// /Chiller_2_Values
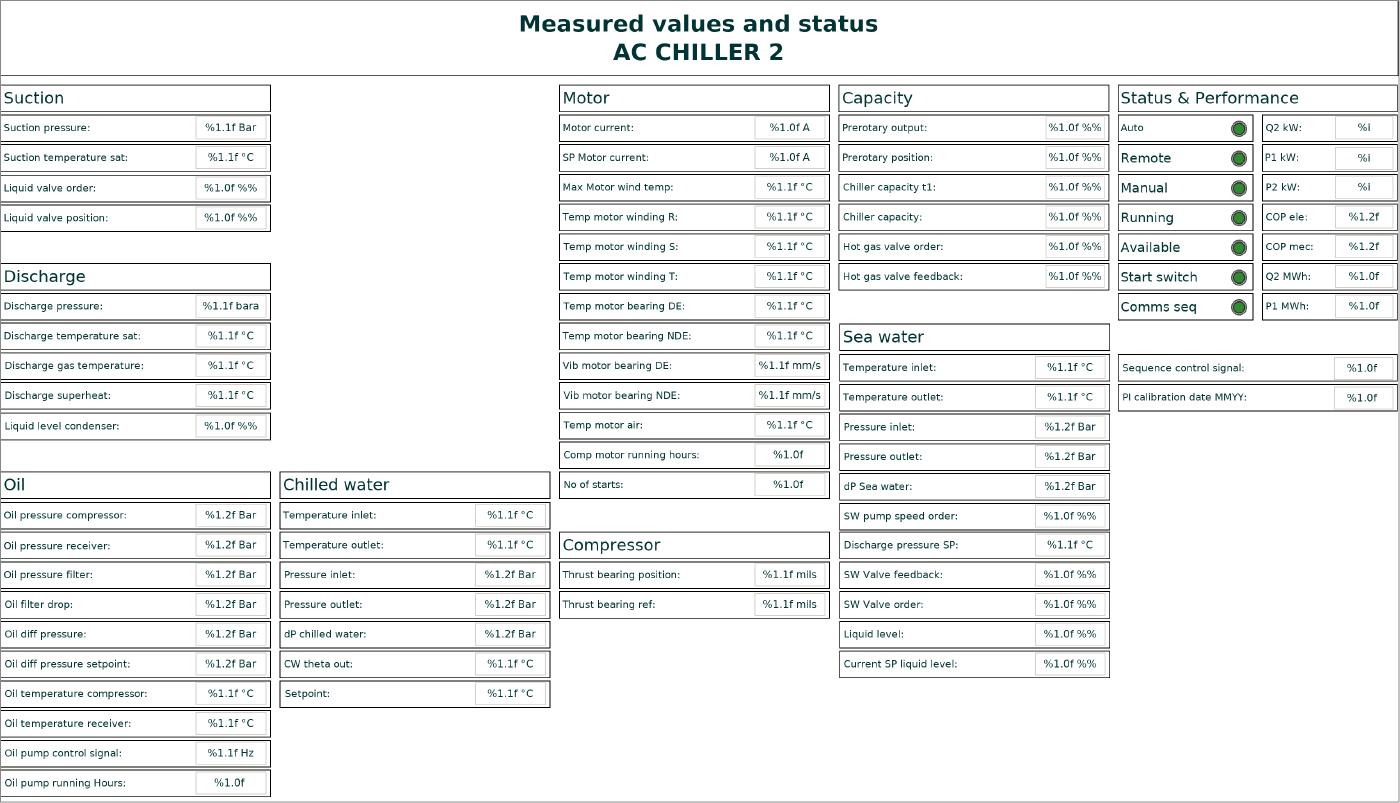
VISUALIZATION Chiller_2_Values  // 1553x891
    Rectangle (0,0 1551x84)
    Label (319,7 912x70), "Measured values and status AC CHILLER 2"
    Rectangle (0,94 300x30)
    Label (1,94 215x30), "Suction"
    Rectangle (0,127 300x30)
    Label (1,122 208x40), "Suction pressure:"
    Textfield (217,129 78x25), "%1.1f Bar", tooltip "Chiller_2.Press_suction_compr", text variable: Chiller_2.Press_suction_compr
        p4168582468: Chiller_2.Press_suction_compr
    Rectangle (0,160 300x30)
    Label (1,155 209x40), "Suction temperature sat:"
    Textfield (217,162 78x25), "%1.1f °C", tooltip "Chiller_2.Suction_saturated_temp", text variable: Chiller_2.Suction_saturated_temp
        p4168582468: Chiller_2.Suction_saturated_temp
    Rectangle (0,194 300x30)
    Label (1,189 211x40), "Liquid valve order:"
    Textfield (217,196 78x25), "%1.0f %%", tooltip "Chiller_2.Liquid_valve_output", text variable: Chiller_2.Liquid_valve_output
        p4168582468: Chiller_2.Liquid_valve_output
    Rectangle (0,227 300x30)
    Label (1,222 216x40), "Liquid valve position:"
    Textfield (217,229 78x25), "%1.0f %%", tooltip "Chiller_2.Feedback_liquid_valve", text variable: Chiller_2.Feedback_liquid_valve
        p4168582468: Chiller_2.Feedback_liquid_valve
    Rectangle (930,94 300x30)
    Label (931,94 162x30), "Capacity"
    Rectangle (930,127 300x30)
    Label (931,126 174x32), "Prerotary output:"
    Textfield (1160,129 65x25), "%1.0f %%", tooltip "Chiller_2.Prerotary_output", text variable: Chiller_2.Prerotary_output
        p4168582468: Chiller_2.Prerotary_output
    Rectangle (930,160 300x30)
    Label (931,159 173x32), "Prerotary position:"
    Textfield (1160,162 65x25), "%1.0f %%", tooltip "Chiller_2.Feedback_PRV", text variable: Chiller_2.Feedback_PRV
        p4168582468: Chiller_2.Feedback_PRV
    Rectangle (930,259 300x30)
    Label (932,258 177x32), "Hot gas valve order:"
    Textfield (1160,261 65x25), "%1.0f %%", tooltip "Chiller_2.Hot_gas_valve_output", text variable: Chiller_2.Hot_gas_valve_output
        p4168582468: Chiller_2.Hot_gas_valve_output
    Rectangle (930,292 300x30)
    Label (932,293 177x28), "Hot gas valve feedback:"
    Textfield (1160,294 65x25), "%1.0f %%", tooltip "Chiller_2.Feedback_HGV", text variable: Chiller_2.Feedback_HGV
        p4168582468: Chiller_2.Feedback_HGV
    Rectangle (0,292 300x30)
    Label (1,292 194x30), "Discharge"
    Rectangle (0,325 300x30)
    Label (1,320 213x40), "Discharge pressure:"
    Textfield (217,327 78x25), "%1.1f bara", tooltip "Chiller_2.Press_discharge_compr", text variable: Chiller_2.Press_discharge_compr
        p4168582468: Chiller_2.Press_discharge_compr
    Rectangle (0,358 300x30)
    Label (1,353 214x40), "Discharge temperature sat:"
    Textfield (217,360 78x25), "%1.1f °C", tooltip "Chiller_2.Discharge_saturated_temp", text variable: Chiller_2.Discharge_saturated_temp
        p4168582468: Chiller_2.Discharge_saturated_temp
    Rectangle (0,391 300x30)
    Label (2,386 213x40), "Discharge gas temperature:"
    Textfield (217,393 78x25), "%1.1f °C", tooltip "Chiller_2.Temp_discharge", text variable: Chiller_2.Temp_discharge
        p4168582468: Chiller_2.Temp_discharge
    Rectangle (0,458 300x30)
    Textfield (217,460 78x25), "%1.0f %%", tooltip "Chiller_2.Liquid_level_condenser", text variable: Chiller_2.Liquid_level_condenser
        p4168582468: Chiller_2.Liquid_level_condenser
    Rectangle (0,424 300x30)
    Label (2,419 212x40), "Discharge superheat:"
    Textfield (217,426 78x25), "%1.1f °C", tooltip "Chiller_2.Discharge_superheat", text variable: Chiller_2.Discharge_superheat
        p4168582468: Chiller_2.Discharge_superheat
    Label (2,453 210x40), "Liquid level condenser:"
    Rectangle (930,193 300x30)
    Label (932,192 174x32), "Chiller capacity t1:"
    Textfield (1160,195 65x25), "%1.0f %%", tooltip "Chiller_2.Chiller_capacity_t1", text variable: Chiller_2.Chiller_capacity_t1
        p4168582468: Chiller_2.Chiller_capacity_t1
    Rectangle (620,94 300x30)
    Label (621,94 194x30), "Motor"
    Rectangle (620,127 300x30)
    Label (621,122 209x40), "Motor current:"
    Textfield (837,129 78x25), "%1.0f A", tooltip "Chiller_2.Motor_current", text variable: Chiller_2.Motor_current
        p4168582468: Chiller_2.Motor_current
    Rectangle (620,226 300x30)
    Label (621,221 210x40), "Temp motor winding R:"
    Textfield (837,228 78x25), "%1.1f °C", tooltip "Chiller_2.Temp_motor_wind_R", text variable: Chiller_2.Temp_motor_wind_R
        p4168582468: Chiller_2.Temp_motor_wind_R
    Rectangle (620,259 300x30)
    Label (622,254 204x40), "Temp motor winding S:"
    Textfield (837,261 78x25), "%1.1f °C", tooltip "Chiller_2.Temp_motor_wind_S", text variable: Chiller_2.Temp_motor_wind_S
        p4168582468: Chiller_2.Temp_motor_wind_S
    Rectangle (620,292 300x30)
    Label (622,287 206x40), "Temp motor winding T:"
    Textfield (837,294 78x25), "%1.1f °C", tooltip "Chiller_2.Temp_motor_wind_T", text variable: Chiller_2.Temp_motor_wind_T
        p4168582468: Chiller_2.Temp_motor_wind_T
    Rectangle (620,325 300x30)
    Label (622,320 216x40), "Temp motor bearing DE:"
    Textfield (837,327 78x25), "%1.1f °C", tooltip "Chiller_2.Temp_motor_bearing_DE", text variable: Chiller_2.Temp_motor_bearing_DE
        p4168582468: Chiller_2.Temp_motor_bearing_DE
    Rectangle (620,358 300x30)
    Label (621,353 218x40), "Temp motor bearing NDE:"
    Textfield (837,360 78x25), "%1.1f °C", tooltip "Chiller_2.Temp_motor_bearing_NDE", text variable: Chiller_2.Temp_motor_bearing_NDE
        p4168582468: Chiller_2.Temp_motor_bearing_NDE
    Rectangle (620,391 300x30)
    Label (621,386 215x40), "Vib motor bearing DE:"
    Textfield (837,393 78x25), "%1.1f mm/s", tooltip "Chiller_2.Vibration_compressor_DE", text variable: Chiller_2.Vibration_compressor_DE
        p4168582468: Chiller_2.Vibration_compressor_DE
    Rectangle (620,424 300x30)
    Label (622,419 215x40), "Vib motor bearing NDE:"
    Textfield (837,426 78x25), "%1.1f mm/s", tooltip "Chiller_2.Vibration_compressor_NDE", text variable: Chiller_2.Vibration_compressor_NDE
        p4168582468: Chiller_2.Vibration_compressor_NDE
    Rectangle (620,457 300x30)
    Label (622,452 210x40), "Temp motor air:"
    Textfield (837,459 78x25), "%1.1f °C", tooltip "Chiller_2.Temp_motor_air", text variable: Chiller_2.Temp_motor_air
        p4168582468: Chiller_2.Temp_motor_air
    Rectangle (620,490 300x30)
    Label (622,485 214x40), "Comp motor running hours:"
    Textfield (837,492 78x25), "%1.0f", tooltip "Chiller_2.Running_hours_compressormotor", text variable: Chiller_2.Running_hours_compressormotor
        p4168582468: Chiller_2.Running_hours_compressormotor
    Rectangle (620,523 300x30)
    Label (622,518 207x40), "No of starts:"
    Textfield (837,525 78x25), "%1.0f", tooltip "Chiller_2.Number_of_starts", text variable: Chiller_2.Number_of_starts
        p4168582468: Chiller_2.Number_of_starts
    Rectangle (310,523 300x30)
    Label (311,523 194x30), "Chilled water"
    Rectangle (310,557 300x30)
    Label (311,552 204x40), "Temperature inlet:"
    Textfield (527,559 78x25), "%1.1f °C", tooltip "Chiller_2.Temp_chilled_medium_in", text variable: Chiller_2.Temp_chilled_medium_in
        p4168582468: Chiller_2.Temp_chilled_medium_in
    Rectangle (310,590 300x30)
    Label (311,585 209x40), "Temperature outlet:"
    Textfield (527,592 78x25), "%1.1f °C", tooltip "Chiller_2.Temp_chilled_medium_out", text variable: Chiller_2.Temp_chilled_medium_out
        p4168582468: Chiller_2.Temp_chilled_medium_out
    Rectangle (310,623 300x30)
    Label (312,618 206x40), "Pressure inlet:"
    Textfield (527,625 78x25), "%1.2f Bar", tooltip "Chiller_2.Press_chilled_medium_in", text variable: Chiller_2.Press_chilled_medium_in
        p4168582468: Chiller_2.Press_chilled_medium_in
    Rectangle (310,656 300x30)
    Label (312,651 208x40), "Pressure outlet:"
    Textfield (527,658 78x25), "%1.2f Bar", tooltip "Chiller_2.Press_chilled_medium_out", text variable: Chiller_2.Press_chilled_medium_out
        p4168582468: Chiller_2.Press_chilled_medium_out
    Rectangle (310,689 300x30)
    Label (312,684 207x40), "dP chilled water:"
    Textfield (527,691 78x25), "%1.2f Bar", tooltip "Chiller_2.dP_CW", text variable: Chiller_2.dP_CW
        p4168582468: Chiller_2.dP_CW
    Rectangle (310,722 300x30)
    Label (312,717 205x40), "CW theta out:"
    Textfield (527,724 78x25), "%1.1f °C", tooltip "Chiller_2.Theta_out", text variable: Chiller_2.Theta_out
        p4168582468: Chiller_2.Theta_out
    Rectangle (310,755 300x30)
    Label (313,750 205x40), "Setpoint:"
    Textfield (527,757 78x25), "%1.1f °C", tooltip "Chiller_2.SP_CW_controller", text variable: Chiller_2.SP_CW_controller
        p4168582468: Chiller_2.SP_CW_controller
    Rectangle (620,160 300x30)
    Label (621,155 209x40), "SP Motor current:"
    Textfield (837,162 78x25), "%1.0f A", tooltip "Chiller_2.SP_MC_controller", text variable: Chiller_2.SP_MC_controller
        p4168582468: Chiller_2.SP_MC_controller
    Rectangle (620,590 300x30)
    Label (621,590 194x30), "Compressor"
    Rectangle (620,623 300x30)
    Label (621,622 216x32), "Thrust bearing position:"
    Textfield (837,625 78x25), "%1.1f mils", tooltip "Chiller_2.Thrust_bearing_position", text variable: Chiller_2.Thrust_bearing_position
        p4168582468: Chiller_2.Thrust_bearing_position
    Rectangle (620,656 300x30)
    Label (621,655 216x32), "Thrust bearing ref:"
    Textfield (837,658 78x25), "%1.1f mils", tooltip "Chiller_2.Proximitor_thrust_pos", text variable: Chiller_2.Proximitor_thrust_pos
        p4168582468: Chiller_2.Proximitor_thrust_pos
    Rectangle (0,523 300x30)
    Label (1,523 194x30), "Oil"
    Rectangle (0,557 300x30)
    Label (1,552 211x40), "Oil pressure compressor:"
    Textfield (217,559 78x25), "%1.2f Bar", tooltip "Chiller_2.Press_oil_compr", text variable: Chiller_2.Press_oil_compr
        p4168582468: Chiller_2.Press_oil_compr
    Rectangle (0,590 300x30)
    Label (1,586 210x40), "Oil pressure receiver:"
    Textfield (217,592 78x25), "%1.2f Bar", tooltip "Chiller_2.Press_oil_receiver", text variable: Chiller_2.Press_oil_receiver
        p4168582468: Chiller_2.Press_oil_receiver
    Rectangle (0,656 300x30)
    Label (2,651 209x40), "Oil filter drop:"
    Textfield (217,658 78x25), "%1.2f Bar", tooltip "Chiller_2.Oil_Filter_Drop", text variable: Chiller_2.Oil_Filter_Drop
        p4168582468: Chiller_2.Oil_Filter_Drop
    Rectangle (0,689 300x30)
    Label (2,684 211x40), "Oil diff pressure:"
    Textfield (217,691 78x25), "%1.2f Bar", tooltip "Chiller_2.Oil_diff_pressure", text variable: Chiller_2.Oil_diff_pressure
        p4168582468: Chiller_2.Oil_diff_pressure
    Rectangle (0,755 300x30)
    Label (2,758 218x24), "Oil temperature compressor:"
    Textfield (217,757 78x25), "%1.1f °C", tooltip "Chiller_2.Temp_oil_inlet_compr", text variable: Chiller_2.Temp_oil_inlet_compr
        p4168582468: Chiller_2.Temp_oil_inlet_compr
    Rectangle (0,788 300x30)
    Label (2,783 210x40), "Oil temperature receiver:"
    Textfield (217,790 78x25), "%1.1f °C", tooltip "Chiller_2.Oil_temp_receiver", text variable: Chiller_2.Oil_temp_receiver
        p4168582468: Chiller_2.Oil_temp_receiver
    Rectangle (0,821 300x30)
    Label (2,816 212x40), "Oil pump control signal:"
    Textfield (217,823 78x25), "%1.1f Hz", tooltip "Chiller_2.Setpoint_conv_oil_pump", text variable: Chiller_2.Setpoint_conv_oil_pump
        p4168582468: Chiller_2.Setpoint_conv_oil_pump
    Rectangle (0,854 300x30)
    Label (2,849 206x40), "Oil pump running Hours:"
    Textfield (217,856 78x25), "%1.0f", tooltip "Chiller_2.Oil_pump_running_hours", text variable: Chiller_2.Oil_pump_running_hours
        p4168582468: Chiller_2.Oil_pump_running_hours
    Rectangle (0,623 300x30)
    Label (1,618 210x40), "Oil pressure filter:"
    Textfield (217,625 78x25), "%1.2f Bar", tooltip "Chiller_2.Oil_pressure_before_filter", text variable: Chiller_2.Oil_pressure_before_filter
        p4168582468: Chiller_2.Oil_pressure_before_filter
    Rectangle (0,722 300x30)
    Label (2,724 211x26), "Oil diff pressure setpoint:"
    Textfield (217,724 78x25), "%1.2f Bar", tooltip "Chiller_2.SP_oil_pressure", text variable: Chiller_2.SP_oil_pressure
        p4168582468: Chiller_2.SP_oil_pressure
    Rectangle (620,193 300x30)
    Label (621,188 210x40), "Max Motor wind temp:"
    Textfield (837,195 78x25), "%1.1f °C", tooltip "Chiller_2.Max_motor_wind_temp", text variable: Chiller_2.Max_motor_wind_temp
        p4168582468: Chiller_2.Max_motor_wind_temp
    Rectangle (931,359 300x30)
    Label (932,359 194x30), "Sea water"
    Rectangle (931,393 300x30)
    Label (932,388 211x40), "Temperature inlet:"
    Textfield (1148,395 78x25), "%1.1f °C", tooltip "Chiller_2.Temp_water_inlet_cond", text variable: Chiller_2.Temp_water_inlet_cond
        p4168582468: Chiller_2.Temp_water_inlet_cond
    Rectangle (931,459 300x30)
    Label (933,454 210x40), "Pressure inlet:"
    Textfield (1148,461 78x25), "%1.2f Bar", tooltip "Chiller_2.Press_water_cond_inlet", text variable: Chiller_2.Press_water_cond_inlet
        p4168582468: Chiller_2.Press_water_cond_inlet
    Rectangle (931,492 300x30)
    Label (933,487 210x40), "Pressure outlet:"
    Textfield (1148,494 78x25), "%1.2f Bar", tooltip "Chiller_2.Press_water_cond_out", text variable: Chiller_2.Press_water_cond_out
        p4168582468: Chiller_2.Press_water_cond_out
    Rectangle (931,525 300x30)
    Label (933,520 210x40), "dP Sea water:"
    Textfield (1148,527 78x25), "%1.2f Bar", tooltip "Chiller_2.dP_CW", text variable: Chiller_2.dP_SW
        p4168582468: Chiller_2.dP_SW
    Rectangle (931,558 300x30)
    Label (933,553 216x40), "SW pump speed order:"
    Textfield (1148,560 78x25), "%1.0f %%", tooltip "Chiller_2.SW_pump_speed_order", text variable: Chiller_2.SW_pump_speed_order
        p4168582468: Chiller_2.SW_pump_speed_order
    Rectangle (931,426 300x30)
    Label (932,421 211x40), "Temperature outlet:"
    Textfield (1148,428 78x25), "%1.1f °C", tooltip "Chiller_2.Temp_water_outlet_cond", text variable: Chiller_2.Temp_water_outlet_cond
        p4168582468: Chiller_2.Temp_water_outlet_cond
    Rectangle (931,590 300x30)
    Label (933,585 208x40), "Discharge pressure SP:"
    Textfield (1148,592 78x25), "%1.1f °C", tooltip "Chiller_2.SP_PID_seawater", text variable: Chiller_2.SP_PID_seawater
        p4168582468: Chiller_2.SP_PID_seawater
    Rectangle (931,623 300x30)
    Label (933,618 208x40), "SW Valve feedback:"
    Textfield (1148,625 78x25), "%1.0f %%", tooltip "Chiller_2.Feedback_seawater_valve_overboard", text variable: Chiller_2.Feedback_seawater_valve_overboard
        p4168582468: Chiller_2.Feedback_seawater_valve_overboard
    Rectangle (931,689 300x30)
    Label (933,684 208x40), "Liquid level:"
    Textfield (1148,691 78x25), "%1.0f %%", tooltip "Chiller_2.Liquid_level_condenser", text variable: Chiller_2.Liquid_level_condenser
        p4168582468: Chiller_2.Liquid_level_condenser
    Rectangle (931,722 300x30)
    Label (933,717 208x40), "Current SP liquid level:"
    Textfield (1148,724 78x25), "%1.0f %%", tooltip "Chiller_2.SP_PID_Level", text variable: Chiller_2.SP_PID_Level
        p4168582468: Chiller_2.SP_PID_Level
    Rectangle (930,226 300x30)
    Label (932,225 174x32), "Chiller capacity:"
    Textfield (1160,228 65x25), "%1.0f %%", tooltip "Chiller_2.Chiller_capacity", text variable: Chiller_2.Chiller_capacity
        p4168582468: Chiller_2.Chiller_capacity
    Rectangle (1240,127 150x30)
    Rectangle (1240,160 150x30)
    Rectangle (1240,193 150x30)
    Rectangle (1240,226 150x30)
    Rectangle (1240,259 150x30)
    Rectangle (1240,292 150x30)
    Rectangle (1240,325 150x30)
    Lamp1 (1363,133 23x20), tooltip "Chiller_2.Unit_auto", variable: Chiller_2.Unit_auto, style: Lamp-Lamp1-Green
    Label (1240,129 112x26), "Auto"
    Label (1240,165 105x21), "Remote"
    Lamp1 (1363,166 23x20), tooltip "Chiller_2.Unit_remote", variable: Chiller_2.Unit_remote, style: Lamp-Lamp1-Green
    Label (1240,198 105x21), "Manual"
    Lamp1 (1363,199 23x20), tooltip "Chiller_2.Unit_manual", variable: Chiller_2.Unit_manual, style: Lamp-Lamp1-Green
    Label (1240,231 105x21), "Running"
    Lamp1 (1363,232 23x20), tooltip "Chiller_2.Unit_running", variable: Chiller_2.Unit_running, style: Lamp-Lamp1-Green
    Label (1240,264 105x21), "Available"
    Lamp1 (1363,265 23x20), tooltip "Chiller_2.Unit_available", variable: Chiller_2.Unit_available, style: Lamp-Lamp1-Green
    Label (1240,297 130x21), "Start switch"
    Lamp1 (1363,298 23x20), tooltip "Chiller_2.Unit_start_switch", variable: Chiller_2.Unit_start_switch, style: Lamp-Lamp1-Green
    Lamp1 (1363,331 23x20), tooltip "Sequence.A_Comms_Chiller_2", variable: Sequence.A_Comms_Chiller_2, style: Lamp-Lamp1-Green
    Label (1240,330 111x21), "Comms seq"
    Rectangle (1240,393 310x30)
    Label (1242,399 227x19), "Sequence control signal:"
    Textfield (1480,396 65x25), "%1.0f", tooltip "Sequence.Seq_cap_order_C2", text variable: Sequence.Seq_cap_order_C2
        p4168582468: Sequence.Seq_cap_order_C2
    Rectangle (1240,426 310x30)
    Label (1242,429 227x24), "PI calibration date MMYY:"
    Textfield (1480,429 65x25), "%1.0f", tooltip "Sequence.Cal_date_ch_2_MMYY", text variable: Sequence.Cal_date_ch_2_MMYY
        p4168582468: Sequence.Cal_date_ch_2_MMYY
    Rectangle (1240,94 310x30)
    Label (1240,94 252x30), "Status & Performance"
    Rectangle (1400,226 150x30)
    Rectangle (1400,127 150x30)
    Rectangle (1400,193 150x30)
    Rectangle (1400,160 150x30)
    Rectangle (1400,292 150x30)
    Rectangle (1400,259 150x30)
    Rectangle (1400,325 150x30)
    Label (1401,228 112x26), "COP ele:"
    Label (1401,126 112x32), "Q2 kW:"
    Label (1401,194 112x28), "P2 kW:"
    Label (1400,159 112x32), "P1 kW:"
    Label (1401,293 112x28), "Q2 MWh:"
    Label (1401,261 112x26), "COP mec:"
    Label (1401,327 112x26), "P1 MWh:"
    Textfield (1481,228 64x25), "%1.2f", tooltip "Sequence.COP_Chiller_2_ele", text variable: Sequence.COP_Chiller_2_ele
        p4168582468: Sequence.COP_Chiller_2_ele
    Textfield (1481,129 64x25), "%i", tooltip "Sequence.Q2kW_Chiller_2", text variable: Sequence.Q2kW_Chiller_2
        p4168582468: Sequence.Q2kW_Chiller_2
    Textfield (1481,195 64x25), "%i", tooltip "Sequence.P2_mot_2_kW", text variable: Sequence.P2_mot_2_kW
        p4168582468: Sequence.P2_mot_2_kW
    Textfield (1481,163 64x25), "%i", tooltip "Sequence.P1_motor_2_kW", text variable: Sequence.P1_motor_2_kW
        p4168582468: Sequence.P1_motor_2_kW
    Textfield (1481,294 64x25), "%1.0f", tooltip "Sequence.Chiller_2_Q2_MWh", text variable: Sequence.Chiller_2_Q2_MWh
        p4168582468: Sequence.Chiller_2_Q2_MWh
    Textfield (1481,261 64x25), "%1.2f", tooltip "Sequence.COP_ch_2_mec", text variable: Sequence.COP_ch_2_mec
        p4168582468: Sequence.COP_ch_2_mec
    Textfield (1481,327 64x25), "%1.0f", tooltip "Sequence.Chiller_2_P1_MWh", text variable: Sequence.Chiller_2_P1_MWh
        p4168582468: Sequence.Chiller_2_P1_MWh
    Rectangle (931,656 300x30)
    Label (933,651 208x40), "SW Valve order:"
    Textfield (1148,658 78x25), "%1.0f %%", tooltip "Chiller_2.Control_signal_SW_valve", text variable: Chiller_2.Control_signal_SW_valve
        p4168582468: Chiller_2.Control_signal_SW_valve
END_VISUALIZATION

// /Chiller_3_Alarm
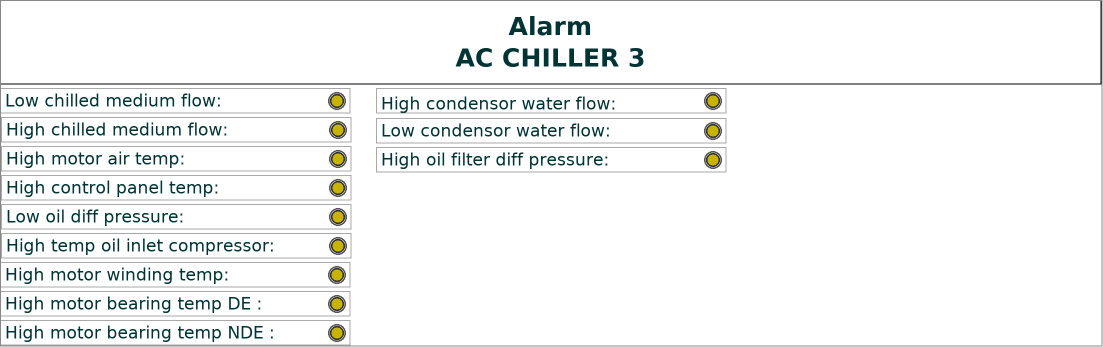
VISUALIZATION Chiller_3_Alarm  // 1103x347
    Rectangle (0,0 1101x84)
    Label (19,7 1063x70), "Alarm AC CHILLER 3"
    Rectangle (1,117 350x25)
    Label (3,119 314x21), "High chilled medium flow:"
    Lamp1 (327,120 22x20), variable: not.Chiller_3.A_High_chilled_medium_flow, style: Lamp-Lamp1-Yellow
    Rectangle (0,262 350x25)
    Label (2,264 314x21), "High motor winding temp:"
    Lamp1 (326,265 22x20), variable: not.Chiller_3.A_High_comp_motor_winding_temp, style: Lamp-Lamp1-Yellow
    Rectangle (0,291 350x25)
    Label (2,293 315x21), "High motor bearing temp DE :"
    Lamp1 (326,294 22x20), variable: not.Chiller_3.A_High_comp_mo_DE_bear_temp, style: Lamp-Lamp1-Yellow
    Rectangle (1,233 350x25)
    Label (3,235 312x21), "High temp oil inlet compressor:"
    Lamp1 (327,236 22x20), variable: not.Chiller_3.A_High_temp_oil_inlet_comp, style: Lamp-Lamp1-Yellow
    Rectangle (1,175 350x25)
    Label (3,177 309x21), "High control panel temp:"
    Lamp1 (327,178 22x20), variable: not.Chiller_3.A_High_control_panel_temp, style: Lamp-Lamp1-Yellow
    Rectangle (1,204 350x25)
    Label (3,206 315x21), "Low oil diff pressure:"
    Lamp1 (327,207 22x20), variable: not.Chiller_3.A_Low_oil_diff_pressure, style: Lamp-Lamp1-Yellow
    Rectangle (376,118 350x25)
    Label (378,120 320x21), "Low condensor water flow:"
    Lamp1 (702,121 22x20), variable: not.Chiller_3.A_Low_sea_water_flow, style: Lamp-Lamp1-Yellow
    Rectangle (376,147 350x25)
    Label (378,149 319x21), "High oil filter diff pressure:"
    Lamp1 (702,150 22x20), variable: not.Chiller_3.A_High_oil_filter_diff_press, style: Lamp-Lamp1-Yellow
    Rectangle (1,146 350x25)
    Label (3,148 314x21), "High motor air temp:"
    Lamp1 (327,149 22x20), variable: not.Chiller_3.A_High_motor_air_temp, style: Lamp-Lamp1-Yellow
    Rectangle (0,320 350x25)
    Label (2,322 315x21), "High motor bearing temp NDE :"
    Lamp1 (326,323 22x20), variable: not.Chiller_3.A_High_comp_mo_NDE_bear_temp, style: Lamp-Lamp1-Yellow
    Rectangle (0,88 350x25)
    Label (2,90 314x21), "Low chilled medium flow:"
    Lamp1 (326,91 22x20), variable: not.Chiller_3.A_Low_chilled_medium_flow, style: Lamp-Lamp1-Yellow
    Rectangle (376,88 350x25)
    Label (378,96 319x15), "High condensor water flow:"
    Lamp1 (702,91 22x20), variable: not.Chiller_3.A_High_condenser_flow, style: Lamp-Lamp1-Yellow
END_VISUALIZATION

// /Chiller_3_Flow_Diagram
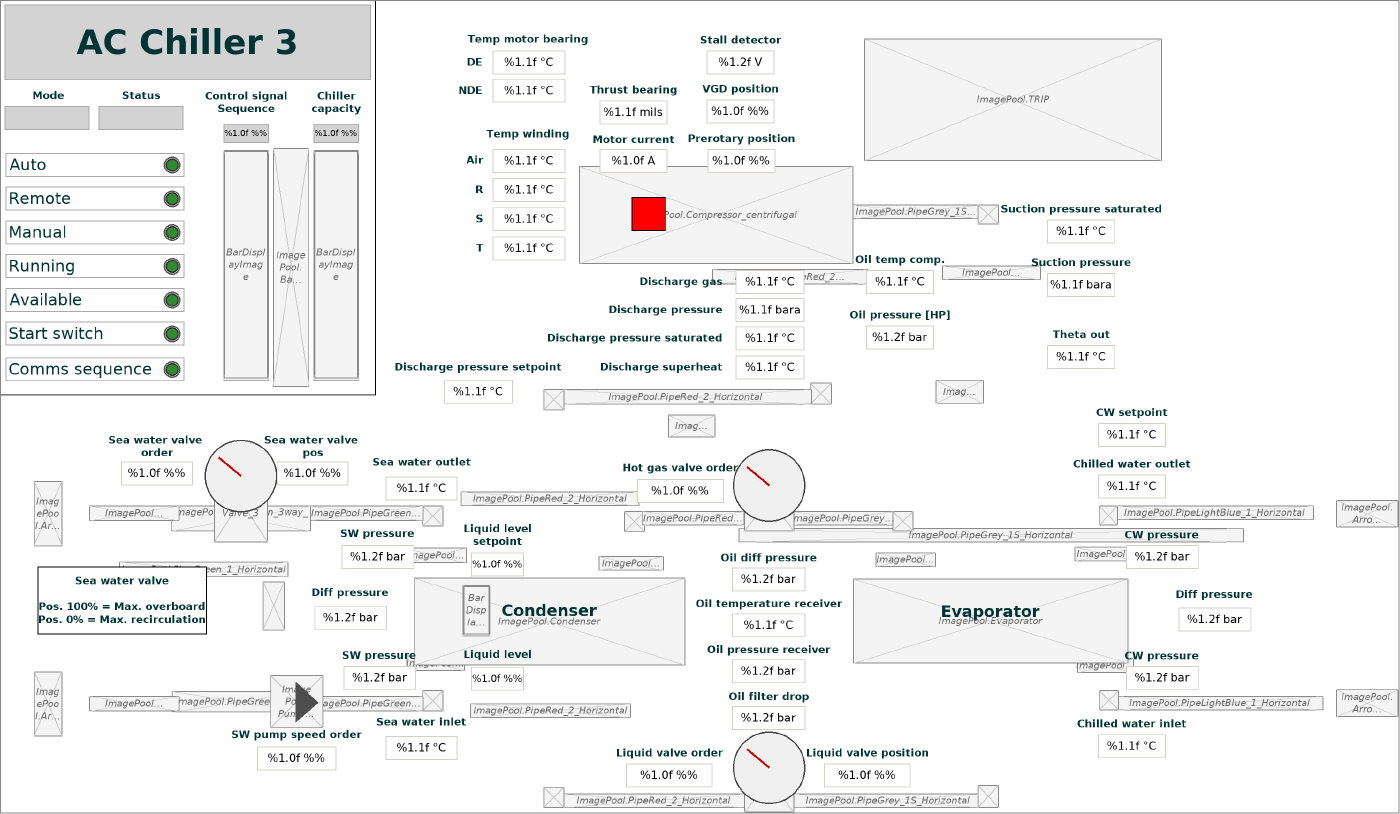
VISUALIZATION Chiller_3_Flow_Diagram  // 1492x868
    Rectangle (0,0 400x421)
    Textfield (238,132 48x20), "%1.0f %%", text variable: Sequence.Seq_cap_order_C3
        p4168582468: Sequence.Seq_cap_order_C3
    Image (1148,702 60x15), angle 270, image: ImagePool.PipeLightBlue_1_Horizontal
    Image (1145,583 67x15), angle 270, image: ImagePool.PipeLightBlue_1_Horizontal
    Image (908,218 137x15), image: ImagePool.PipeGrey_1S_Horizontal
    Image (845,846 202x15), image: ImagePool.PipeGrey_1S_Horizontal
    Image (933,589 64x15), angle 270, image: ImagePool.PipeGrey_1S_Horizontal
    Image (787,563 538x15), angle 270, image: ImagePool.PipeGrey_1S_Horizontal
    Image (843,545 110x15), image: ImagePool.PipeGrey_1S_Horizontal
    Image (638,593 69x15), angle 270, image: ImagePool.PipeRed_2_Horizontal
    Image (501,750 171x15), angle 270, image: ImagePool.PipeRed_2_Horizontal
    Label (218,94 89x30), "Control signal Sequence"
    Image (617,177 292x104), image: ImagePool.Compressor_centrifugal
    Image (759,287 166x16), angle 270, image: ImagePool.PipeRed_2_Horizontal
    Image (863,408 23x23), image: ImagePool.PipeRed_2_LU
    Image (596,415 269x16), image: ImagePool.PipeRed_2_Horizontal
    Image (909,617 293x90), image: ImagePool.Evaporator
    Image (431,584 66x16), angle 270, image: ImagePool.PipeGreen_1_Horizontal
    Image (450,539 22x22), image: ImagePool.PipeGreen_1_LD
    Image (329,539 122x16), image: ImagePool.PipeGreen_1_Horizontal
    Label (331,617 84x30), "Diff pressure"
    Textfield (335,646 77x25), "%1.2f bar", text variable: Chiller_3.dP_SW
        p4168582468: Chiller_3.dP_SW
    Image (127,599 180x16), angle 270, image: ImagePool.PipeGreen_1_Horizontal
    Image (183,737 147x22), image: ImagePool.PipeGreen_3way
    Image (433,699 62x16), angle 270, image: ImagePool.PipeGreen_1_Horizontal
    Image (450,736 22x22), image: ImagePool.PipeGreen_2_LU
    Image (329,742 122x16), image: ImagePool.PipeGreen_1_Horizontal
    Image (182,539 149x27), image: ImagePool.PipeGreen_3way_2
    Image (228,490 57x88), image: ImagePool.Valve_3
    Image (288,720 56x56), image: ImagePool.Pump_Large_3
    Polygon (315,746) (315,727) (339,749) (315,770) (315,762), colour toggle: Chiller_3.Sea_water_pump
    Image (36,513 30x69), angle 90, image: ImagePool.Arrow green down
    Image (36,716 30x69), angle 270, image: ImagePool.Arrow green down
    Image (579,415 22x22), image: ImagePool.PipeRed_1_RD
    Image (491,524 190x15), angle 270, image: ImagePool.PipeRed_2_Horizontal
    Label (360,554 84x30), "SW pressure"
    Textfield (364,581 77x25), "%1.2f bar", text variable: Chiller_3.Press_water_cond_out
        p4168582468: Chiller_3.Press_water_cond_out
    Image (95,539 96x16), image: ImagePool.PipeGreen_1_Horizontal
    Image (95,742 96x16), image: ImagePool.PipeGreen_1_Horizontal
    Image (441,616 289x93), image: ImagePool.Condenser
    Image (598,846 197x15), image: ImagePool.PipeRed_2_Horizontal
    Image (579,839 22x22), image: ImagePool.PipeRed_2_RU
    Label (362,684 84x30), "SW pressure"
    Textfield (366,710 77x25), "%1.2f bar", text variable: Chiller_3.Press_water_cond_inlet
        p4168582468: Chiller_3.Press_water_cond_inlet
    Image (793,501 53x65), image: ImagePool.Valve_2
    Image (793,801 53x65), image: ImagePool.Valve_2
    Image (665,545 22x22), image: ImagePool.PipeRed_1_RD
    Image (684,545 109x15), image: ImagePool.PipeRed_2_Horizontal
    Image (951,545 22x21), image: ImagePool.PipeGrey_2_LD
    Image (1042,837 22x24), image: ImagePool.PipeGrey_3_LU
    Image (1042,218 22x21), image: ImagePool.PipeGrey_2_LD
    Image (1004,283 105x15), angle 270, image: ImagePool.PipeGrey_1S_Horizontal
    Label (521,636 129x30), "Condenser"
    Label (991,637 129x30), "Evaporator"
    Image (1189,539 211x15), image: ImagePool.PipeLightBlue_1_Horizontal
    Image (1171,539 20x21), image: ImagePool.PipeLightBlue_3_RD
    Image (1190,742 220x15), image: ImagePool.PipeLightBlue_1_Horizontal
    Image (1171,736 21x21), image: ImagePool.PipeLightBlue_3_RU
    Image (1424,533 66x29), angle 180, image: ImagePool.Arrow lightblue left
    Image (1424,735 66x29), image: ImagePool.Arrow lightblue left
    Image (280,620 23x52), image: ImagePool.Arrow green down
    Image (712,442 50x24), image: ImagePool.Arrow red left
    Image (997,405 51x25), angle 90, image: ImagePool.Arrow gray left
    Image (291,158 38x254), image: ImagePool.BarScale3
    Label (324,94 69x30), "Chiller capacity"
    Textfield (105,113 90x25), text list: 'TextList_PT', text index: Chiller_3.Unit_switch_status
    Textfield (5,113 90x25), text list: 'TextList_PT', text index: Chiller_3.Unit_start_switch
    Textfield (334,132 48x20), "%1.0f %%", text variable: Chiller_3.Chiller_capacity_t1
        p4168582468: Chiller_3.Chiller_capacity_t1
    Textfield (5,5 390x80), "AC Chiller 3"
    Textfield (679,511 92x25), "%1.0f %%", text variable: Chiller_3.Hot_gas_valve_output
        p4168582468: Chiller_3.Hot_gas_valve_output
    Label (664,484 122x30), "Hot gas valve order"
    Meter360 (781,479 77x77), value: Chiller_3.Feedback_HGV, style: Meter-Meter360-Gray, scale format: %1.0f, scale 0..100
        p3451962224: ImagePool.Invisible
    Meter360 (781,780 77x77), value: Chiller_3.Feedback_liquid_valve, style: Meter-Meter360-Gray, scale format: %1.0f, scale 0..100
        p3451962224: ImagePool.Invisible
    Meter360 (218,469 77x77), value: Chiller_3.Feedback_sea_water_valve, style: Meter-Meter360-Gray, scale format: %1.0f, scale 0..100
        p3451962224: ImagePool.Invisible
    Textfield (502,589 56x25), "%1.0f %%", text variable: Chiller_3.SP_PID_Level
        p4168582468: Chiller_3.SP_PID_Level
    Label (494,551 73x39), "Liquid level setpoint"
    Textfield (502,711 56x25), "%1.0f %%", text variable: Chiller_3.Liquid_level_condenser
        p4168582468: Chiller_3.Liquid_level_condenser
    Label (491,683 79x30), "Liquid level"
    Textfield (639,159 72x25), "%1.0f A", text variable: Chiller_3.Motor_current
        p4168582468: Chiller_3.Motor_current
    Label (634,138 83x22), "Motor current"
    Textfield (274,796 84x25), "%1.0f %%", text variable: Chiller_3.SW_pump_speed_order
        p4168582468: Chiller_3.SW_pump_speed_order
    Label (250,770 132x27), "SW pump speed order"
    Textfield (473,405 73x25), "%1.1f °C", tooltip "Chiller_3.SP_PID_seawater", text variable: Chiller_3.SP_PID_seawater
    Textfield (784,348 73x25), "%1.1f °C", text variable: Chiller_3.Discharge_saturated_temp
        p4168582468: Chiller_3.Discharge_saturated_temp
    Label (589,347 184x27), "Discharge pressure saturated"
    Label (425,378 169x27), "Discharge pressure setpoint"
    Textfield (411,785 76x25), "%1.1f °C", text variable: Chiller_3.Temp_water_inlet_cond
        p4168582468: Chiller_3.Temp_water_inlet_cond
    Label (399,755 100x30), "Sea water inlet"
    Label (678,287 95x27), "Discharge gas"
    Textfield (784,288 73x25), "%1.1f °C", text variable: Chiller_3.Temp_discharge
        p4168582468: Chiller_3.Temp_discharge
    Label (644,317 129x27), "Discharge pressure"
    Textfield (784,318 73x25), "%1.1f bara", text variable: Chiller_3.Press_discharge_compr
        p4168582468: Chiller_3.Press_discharge_compr
    Textfield (784,379 73x25), "%1.1f °C", text variable: Chiller_3.Discharge_superheat
        p4168582468: Chiller_3.Discharge_superheat
    Label (589,378 184x27), "Discharge superheat"
    Label (631,84 89x24), "Thrust bearing"
    Textfield (639,107 72x25), "%1.1f mils", text variable: Chiller_3.Thrust_bearing_position
        p4168582468: Chiller_3.Thrust_bearing_position
    Label (115,461 105x30), "Sea water valve order"
    Textfield (129,492 76x25), "%1.0f %%", text variable: Chiller_3.Control_signal_SW_valve
        p4168582468: Chiller_3.Control_signal_SW_valve
    Label (281,461 105x30), "Sea water valve pos"
    Textfield (295,492 76x25), "%1.0f %%", text variable: Chiller_3.Feedback_sea_water_valve
        p4168582468: Chiller_3.Feedback_sea_water_valve
    Label (857,788 135x30), "Liquid valve position"
    Textfield (878,814 92x25), "%1.0f %%", text variable: Chiller_3.Feedback_liquid_valve
        p4168582468: Chiller_3.Feedback_liquid_valve
    Textfield (780,753 78x25), "%1.2f bar", text variable: Chiller_3.Oil_Filter_Drop
        p4168582468: Chiller_3.Oil_Filter_Drop
    Label (778,732 83x22), "Oil filter drop"
    Textfield (667,814 92x25), "%1.0f %%", text variable: Chiller_3.Liquid_valve_output
        p4168582468: Chiller_3.Liquid_valve_output
    Label (646,788 135x30), "Liquid valve order"
    Textfield (780,703 78x25), "%1.2f bar", text variable: Chiller_3.Press_oil_receiver
        p4168582468: Chiller_3.Press_oil_receiver
    Label (752,682 135x22), "Oil pressure receiver"
    Textfield (780,654 78x25), "%1.1f °C", text variable: Chiller_3.Oil_temp_receiver
        p4168582468: Chiller_3.Oil_temp_receiver
    Label (748,633 143x22), "Oil temperature receiver"
    Textfield (780,605 78x25), "%1.2f bar", text variable: Chiller_3.Oil_diff_pressure
        p4168582468: Chiller_3.Oil_diff_pressure
    Label (769,584 101x22), "Oil diff pressure"
    Label (738,136 105x24), "Prerotary position"
    Textfield (754,159 72x25), "%1.0f %%", text variable: Chiller_3.Feedback_PRV
        p4168582468: Chiller_3.Feedback_PRV
    Label (1067,211 171x24), "Suction pressure saturated"
    Textfield (1116,234 72x25), "%1.1f °C", text variable: Chiller_3.Suction_saturated_temp
        p4168582468: Chiller_3.Suction_saturated_temp
    Textfield (1116,291 72x25), "%1.1f bara", text variable: Chiller_3.Press_suction_compr
        p4168582468: Chiller_3.Press_suction_compr
    Label (1067,268 171x24), "Suction pressure"
    Textfield (1116,368 72x25), "%1.1f °C", text variable: Chiller_3.Theta_out
        p4168582468: Chiller_3.Theta_out
    Label (1111,345 83x24), "Theta out"
    Label (1196,557 84x27), "CW pressure"
    Textfield (1200,581 77x25), "%1.2f bar", text variable: Chiller_3.Press_chilled_medium_out
        p4168582468: Chiller_3.Press_chilled_medium_out
    Textfield (1200,710 77x25), "%1.2f bar", text variable: Chiller_3.Press_chilled_medium_in
        p4168582468: Chiller_3.Press_chilled_medium_in
    Label (1196,686 84x27), "CW pressure"
    Textfield (1170,506 72x25), "%1.1f °C", text variable: Chiller_3.Temp_chilled_medium_out
        p4168582468: Chiller_3.Temp_chilled_medium_out
    Label (1146,483 121x24), "Chilled water outlet"
    Label (1146,428 121x24), "CW setpoint"
    Textfield (1170,451 72x25), "%1.1f °C", text variable: Chiller_3.SP_PID_compressor
        p4168582468: Chiller_3.SP_PID_compressor
    Label (1252,619 84x30), "Diff pressure"
    Textfield (1256,648 77x25), "%1.2f bar", text variable: Chiller_3.dP_CW
        p4168582468: Chiller_3.dP_CW
    Textfield (1170,783 72x25), "%1.1f °C", text variable: Chiller_3.Temp_chilled_medium_in
        p4168582468: Chiller_3.Temp_chilled_medium_in
    Label (1146,760 121x24), "Chilled water inlet"
    Group (6,271 190x25)
        Rectangle (0,0 190x25)
        Label (0,2 105x21), "Running"
        Lamp1 (166,3 23x20), variable: Chiller_3.Unit_running, style: Lamp-Lamp1-Green
    Group (6,163 190x25)
        Rectangle (0,0 190x25)
        Label (1,2 105x21), "Auto"
        Lamp1 (166,3 23x20), variable: Chiller_3.Unit_auto, style: Lamp-Lamp1-Green
    Group (6,199 190x25)
        Rectangle (0,0 190x25)
        Label (0,2 105x21), "Remote"
        Lamp1 (166,3 23x20), variable: Chiller_3.Unit_remote, style: Lamp-Lamp1-Green
    Group (6,235 190x25)
        Rectangle (0,0 190x25)
        Label (0,2 105x21), "Manual"
        Lamp1 (166,3 23x20), variable: Chiller_3.Unit_manual, style: Lamp-Lamp1-Green
    Group (6,307 190x25)
        Rectangle (0,0 190x25)
        Label (1,2 105x21), "Available"
        Lamp1 (166,3 23x20), variable: Chiller_3.Unit_available, style: Lamp-Lamp1-Green
    Group (6,343 190x25)
        Rectangle (0,0 190x25)
        Label (0,2 130x21), "Start switch"
        Lamp1 (166,3 23x20), variable: Chiller_3.Unit_start_switch, style: Lamp-Lamp1-Green
    Group (6,381 190x25)
        Rectangle (0,0 190x25)
        Label (0,2 160x21), "Comms sequence"
        Lamp1 (166,3 23x20), variable: Sequence.A_Comms_Chiller_3, style: Lamp-Lamp1-Green
    Label (912,265 95x24), "Oil temp comp."
    Textfield (923,288 72x25), "%1.1f °C", text variable: Chiller_3.Temp_oil_inlet_compr
        p4168582468: Chiller_3.Temp_oil_inlet_compr
    Label (902,324 115x24), "Oil pressure [HP]"
    Textfield (923,347 72x25), "%1.2f bar", text variable: Chiller_3.Press_oil_compr
        p4168582468: Chiller_3.Press_oil_compr
    Image (921,41 317x130), invisible if: Chiller_3.Unit_alarm, image: ImagePool.ALARM
    Image (921,41 317x130), invisible if: Chiller_3.Unit_trip, image: ImagePool.TRIP
    Label (7,87 89x30), "Mode"
    Label (106,87 89x30), "Status"
    Rectangle (334,160 48x246)
    Image (238,160 48x246), image: ImagePool.CapBarTranparant
    BarDisplayImage (239,161 46x242), value: Sequence.Seq_cap_order_C3, style: BarDisplayImage-Gray, scale format: %.0f, scale 0..100
        p3451962224: ImagePool.Invisible
    Image (334,160 48x246), image: ImagePool.CapBarTranparant
    BarDisplayImage (335,161 46x242), value: Chiller_3.Chiller_capacity_t1, style: BarDisplayImage-Gray, scale format: %.0f, scale 0..100
        p3451962224: ImagePool.Invisible
    Group (40,604 180x72)
        Rectangle (0,0 180x72)
        Label (0,0 180x72), "Sea water valve Pos. 100% = Max. overboard Pos. 0% = Max. recirculation"
    Rectangle (493,624 28x52)
    Image (493,624 29x54), image: ImagePool.CapBarTranparant
    BarDisplayImage (494,625 27x51), value: Chiller_3.Liquid_level_condenser, style: BarDisplayImage-Gray, scale format: %.0f, scale 0..100
        p3451962224: ImagePool.Invisible
    Label (746,31 87x24), "Stall detector"
    Textfield (753,54 72x25), "%1.2f V", text variable: Chiller_3.Stall_detector
        p4168582468: Chiller_3.Stall_detector
    Rectangle (673,210 36x36), colour toggle: Chiller_3.Unit_running
    Rectangle (673,210 36x36), colour toggle: Chiller_3.Unit_alarm
    Rectangle (673,210 36x36), colour toggle: Chiller_3.Unit_trip
    Label (500,27 126x30), "Temp motor bearing"
    Textfield (525,84 77x25), "%1.1f °C", text variable: Chiller_3.Temp_motor_bearing_NDE
        p4168582468: Chiller_3.Temp_motor_bearing_NDE
    Textfield (525,54 77x25), "%1.1f °C", text variable: Chiller_3.Temp_motor_bearing_DE
        p4168582468: Chiller_3.Temp_motor_bearing_DE
    Label (480,54 37x25), "DE"
    Label (480,84 37x25), "NDE"
    Label (746,83 87x24), "VGD position"
    Textfield (753,106 72x25), "%1.0f %%", text variable: Chiller_3.Feedback_VGD
        p4168582468: Chiller_3.Feedback_VGD
    Label (521,128 84x30), "Temp winding"
    Textfield (525,190 77x25), "%1.1f °C", text variable: Chiller_3.Temp_motor_wind_R
        p4168582468: Chiller_3.Temp_motor_wind_R
    Label (493,190 25x25), "R"
    Textfield (525,221 77x25), "%1.1f °C", text variable: Chiller_3.Temp_motor_wind_S
        p4168582468: Chiller_3.Temp_motor_wind_S
    Label (493,221 25x25), "S"
    Textfield (525,252 77x25), "%1.1f °C", text variable: Chiller_3.Temp_motor_wind_T
        p4168582468: Chiller_3.Temp_motor_wind_T
    Label (493,252 25x25), "T"
    Label (481,156 37x30), "Air"
    Textfield (525,159 77x25), "%1.1f °C", text variable: Chiller_3.Temp_motor_air
        p4168582468: Chiller_3.Temp_motor_air
    Textfield (411,508 76x25), "%1.1f °C", text variable: Chiller_3.Temp_water_outlet_cond
        p4168582468: Chiller_3.Temp_water_outlet_cond
    Label (397,478 105x30), "Sea water outlet"
END_VISUALIZATION

// /Chiller_3_Flow_Diagram
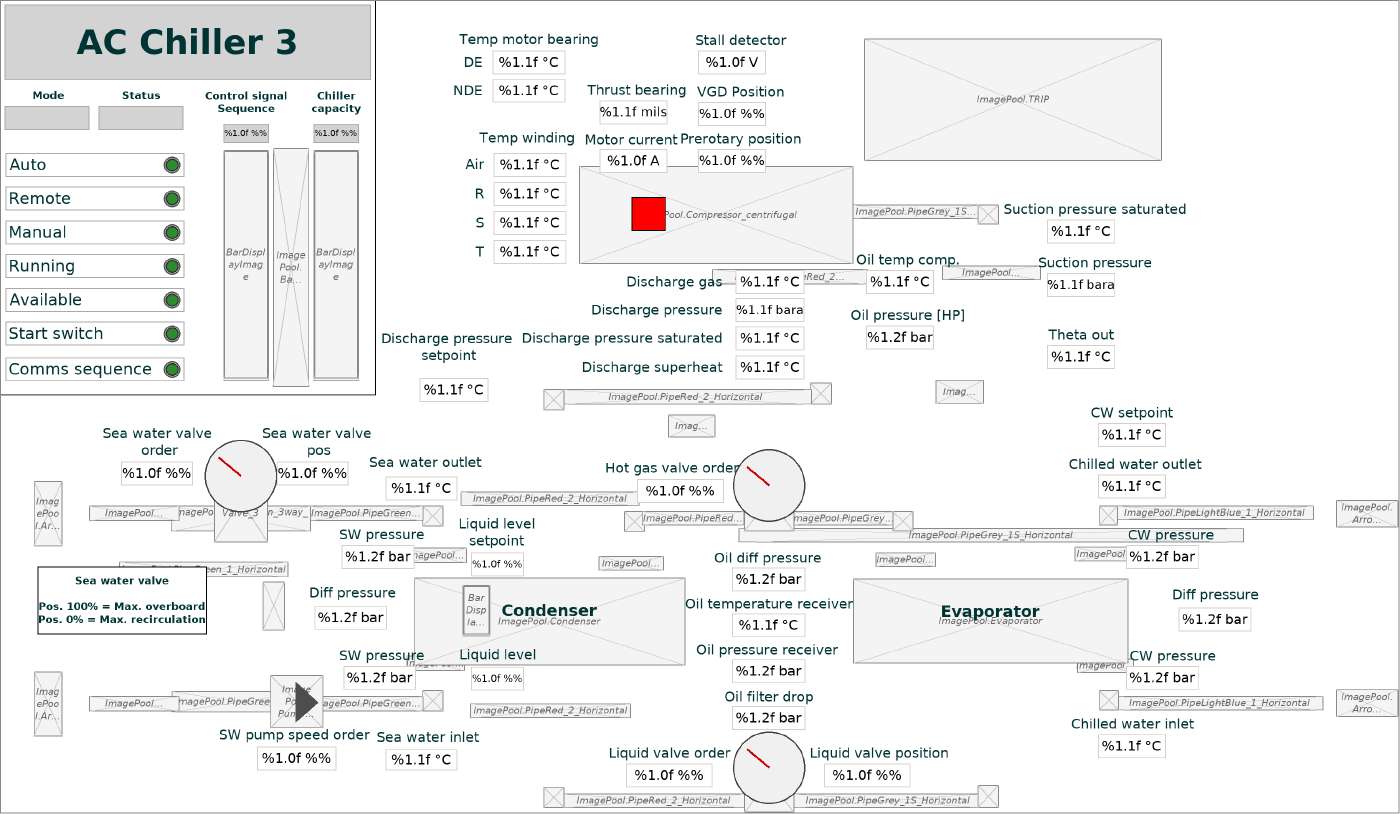
VISUALIZATION Chiller_3_Flow_Diagram  // 1492x868
    Rectangle (0,0 400x421)
    Textfield (238,132 48x20), "%1.0f %%", text variable: Sequence.Seq_cap_order_C1
        p4168582468: Sequence.Seq_cap_order_C1
    Image (1148,702 60x15), angle 270, image: ImagePool.PipeLightBlue_1_Horizontal
    Image (1145,583 67x15), angle 270, image: ImagePool.PipeLightBlue_1_Horizontal
    Image (908,218 137x15), image: ImagePool.PipeGrey_1S_Horizontal
    Image (845,846 202x15), image: ImagePool.PipeGrey_1S_Horizontal
    Image (933,589 64x15), angle 270, image: ImagePool.PipeGrey_1S_Horizontal
    Image (787,563 538x15), angle 270, image: ImagePool.PipeGrey_1S_Horizontal
    Image (843,545 110x15), image: ImagePool.PipeGrey_1S_Horizontal
    Image (638,593 69x15), angle 270, image: ImagePool.PipeRed_2_Horizontal
    Image (501,750 171x15), angle 270, image: ImagePool.PipeRed_2_Horizontal
    Label (218,94 89x30), "Control signal Sequence"
    Image (617,177 292x104), image: ImagePool.Compressor_centrifugal
    Image (759,287 166x16), angle 270, image: ImagePool.PipeRed_2_Horizontal
    Image (863,408 23x23), image: ImagePool.PipeRed_2_LU
    Image (596,415 269x16), image: ImagePool.PipeRed_2_Horizontal
    Image (909,617 293x90), image: ImagePool.Evaporator
    Image (431,584 66x16), angle 270, image: ImagePool.PipeGreen_1_Horizontal
    Image (450,539 22x22), image: ImagePool.PipeGreen_1_LD
    Image (329,539 122x16), image: ImagePool.PipeGreen_1_Horizontal
    Label (311,617 130x30), "Diff pressure"
    Textfield (335,646 77x25), "%1.2f bar", text variable: Chiller_3.dP_SW
        p4168582468: Chiller_3.dP_SW
    Image (127,599 180x16), angle 270, image: ImagePool.PipeGreen_1_Horizontal
    Image (183,737 147x22), image: ImagePool.PipeGreen_3way
    Image (433,699 62x16), angle 270, image: ImagePool.PipeGreen_1_Horizontal
    Image (450,736 22x22), image: ImagePool.PipeGreen_2_LU
    Image (329,742 122x16), image: ImagePool.PipeGreen_1_Horizontal
    Image (182,539 149x27), image: ImagePool.PipeGreen_3way_2
    Image (228,490 57x88), image: ImagePool.Valve_3
    Image (288,720 56x56), image: ImagePool.Pump_Large_3
    Polygon (315,746) (315,727) (339,749) (315,770) (315,762), colour toggle: Chiller_3.Sea_water_pump
    Image (36,513 30x69), angle 90, image: ImagePool.Arrow green down
    Image (36,716 30x69), angle 270, image: ImagePool.Arrow green down
    Image (579,415 22x22), image: ImagePool.PipeRed_1_RD
    Image (491,524 190x15), angle 270, image: ImagePool.PipeRed_2_Horizontal
    Label (342,555 130x30), "SW pressure"
    Textfield (364,581 77x25), "%1.2f bar", text variable: Chiller_3.Press_water_cond_out
        p4168582468: Chiller_3.Press_water_cond_out
    Image (95,539 96x16), image: ImagePool.PipeGreen_1_Horizontal
    Image (95,742 96x16), image: ImagePool.PipeGreen_1_Horizontal
    Image (441,616 289x93), image: ImagePool.Condenser
    Image (598,846 197x15), image: ImagePool.PipeRed_2_Horizontal
    Image (579,839 22x22), image: ImagePool.PipeRed_2_RU
    Label (342,684 130x30), "SW pressure"
    Textfield (366,710 77x25), "%1.2f bar", text variable: Chiller_3.Press_water_cond_inlet
        p4168582468: Chiller_3.Press_water_cond_inlet
    Image (793,501 53x65), image: ImagePool.Valve_2
    Image (793,801 53x65), image: ImagePool.Valve_2
    Image (665,545 22x22), image: ImagePool.PipeRed_1_RD
    Image (684,545 109x15), image: ImagePool.PipeRed_2_Horizontal
    Image (951,545 22x21), image: ImagePool.PipeGrey_2_LD
    Image (1042,837 22x24), image: ImagePool.PipeGrey_3_LU
    Image (1042,218 22x21), image: ImagePool.PipeGrey_2_LD
    Image (1004,283 105x15), angle 270, image: ImagePool.PipeGrey_1S_Horizontal
    Label (521,636 129x30), "Condenser"
    Label (991,637 129x30), "Evaporator"
    Image (1189,539 211x15), image: ImagePool.PipeLightBlue_1_Horizontal
    Image (1171,539 20x21), image: ImagePool.PipeLightBlue_3_RD
    Image (1190,742 220x15), image: ImagePool.PipeLightBlue_1_Horizontal
    Image (1171,736 21x21), image: ImagePool.PipeLightBlue_3_RU
    Image (1424,533 66x29), angle 180, image: ImagePool.Arrow lightblue left
    Image (1424,735 66x29), image: ImagePool.Arrow lightblue left
    Image (280,620 23x52), image: ImagePool.Arrow green down
    Image (712,442 50x24), image: ImagePool.Arrow red left
    Image (997,405 51x25), angle 90, image: ImagePool.Arrow gray left
    Image (291,158 38x254), image: ImagePool.BarScale3
    Label (324,94 69x30), "Chiller capacity"
    Textfield (105,113 90x25), text list: 'TextList_PT', text index: Chiller_3.Unit_switch_status
    Textfield (5,113 90x25), text list: 'TextList_PT', text index: Chiller_3.Unit_start_switch
    Textfield (334,132 48x20), "%1.0f %%", tooltip "Chiller_3.Chiller_capacity", text variable: Chiller_3.Chiller_capacity
        p4168582468: Chiller_3.Chiller_capacity
    Textfield (5,5 390x80), "AC Chiller 3"
    Textfield (679,511 92x25), "%1.0f %%", text variable: Chiller_3.Hot_gas_valve_output
        p4168582468: Chiller_3.Hot_gas_valve_output
    Label (639,484 155x30), "Hot gas valve order"
    Meter360 (781,479 77x77), value: Chiller_3.Feedback_HGV, style: Meter-Meter360-Gray, scale format: %1.0f, scale 0..100
        p3451962224: ImagePool.Invisible
    Meter360 (781,780 77x77), value: Chiller_3.Feedback_liquid_valve, style: Meter-Meter360-Gray, scale format: %1.0f, scale 0..100
        p3451962224: ImagePool.Invisible
    Meter360 (218,469 77x77), value: Chiller_3.Feedback_sea_water_valve, style: Meter-Meter360-Gray, scale format: %1.0f, scale 0..100
        p3451962224: ImagePool.Invisible
    Textfield (502,589 56x25), "%1.0f %%", text variable: Chiller_3.SP_PID_Level
        p4168582468: Chiller_3.SP_PID_Level
    Label (482,545 95x45), "Liquid level setpoint"
    Textfield (502,711 56x25), "%1.0f %%", text variable: Chiller_3.Liquid_level_condenser
        p4168582468: Chiller_3.Liquid_level_condenser
    Label (491,683 79x30), "Liquid level"
    Textfield (639,159 72x25), "%1.0f A", text variable: Chiller_3.Motor_current
        p4168582468: Chiller_3.Motor_current
    Label (617,138 111x22), "Motor current"
    Textfield (274,796 84x25), "%1.0f %%", text variable: Chiller_3.SW_pump_speed_order
        p4168582468: Chiller_3.SW_pump_speed_order
    Label (228,770 172x27), "SW pump speed order"
    Textfield (447,403 73x25), "%1.1f °C", tooltip "Chiller_3.SP_PID_seawater", text variable: Chiller_3.SP_PID_seawater
    Textfield (784,348 73x25), "%1.1f °C", text variable: Chiller_3.Discharge_saturated_temp
        p4168582468: Chiller_3.Discharge_saturated_temp
    Label (552,347 221x27), "Discharge pressure saturated"
    Label (401,339 150x62), "Discharge pressure setpoint"
    Textfield (411,799 76x22), "%1.1f °C", text variable: Chiller_3.Temp_water_inlet_cond
        p4168582468: Chiller_3.Temp_water_inlet_cond
    Label (391,771 130x30), "Sea water inlet"
    Label (646,287 127x27), "Discharge gas"
    Textfield (784,288 73x25), "%1.1f °C", text variable: Chiller_3.Temp_discharge
        p4168582468: Chiller_3.Temp_discharge
    Label (617,317 156x27), "Discharge pressure"
    Textfield (784,318 73x25), "%1.1f bara", text variable: Chiller_3.Press_discharge_compr
        p4168582468: Chiller_3.Press_discharge_compr
    Textfield (784,379 73x25), "%1.1f °C", text variable: Chiller_3.Discharge_superheat
        p4168582468: Chiller_3.Discharge_superheat
    Label (589,378 184x27), "Discharge superheat"
    Label (612,84 134x24), "Thrust bearing"
    Textfield (639,107 72x25), "%1.1f mils", text variable: Chiller_3.Thrust_bearing_position
        p4168582468: Chiller_3.Thrust_bearing_position
    Label (106,451 128x40), "Sea water valve order"
    Textfield (129,492 76x25), "%1.0f %%", text variable: Chiller_3.Control_signal_SW_valve
        p4168582468: Chiller_3.Control_signal_SW_valve
    Label (280,451 120x40), "Sea water valve pos"
    Textfield (295,492 76x25), "%1.0f %%", text variable: Chiller_3.Feedback_sea_water_valve
        p4168582468: Chiller_3.Feedback_sea_water_valve
    Label (857,788 160x30), "Liquid valve position"
    Textfield (878,814 92x25), "%1.0f %%", text variable: Chiller_3.Feedback_liquid_valve
        p4168582468: Chiller_3.Feedback_liquid_valve
    Textfield (780,753 78x25), "%1.2f bar", text variable: Chiller_3.Oil_Filter_Drop
        p4168582468: Chiller_3.Oil_Filter_Drop
    Label (754,732 131x22), "Oil filter drop"
    Textfield (667,814 92x25), "%1.0f %%", text variable: Chiller_3.Liquid_valve_output
        p4168582468: Chiller_3.Liquid_valve_output
    Label (646,788 135x30), "Liquid valve order"
    Textfield (780,703 78x25), "%1.2f bar", text variable: Chiller_3.Press_oil_receiver
        p4168582468: Chiller_3.Press_oil_receiver
    Label (736,682 163x22), "Oil pressure receiver"
    Textfield (780,654 78x25), "%1.1f °C", text variable: Chiller_3.Oil_temp_receiver
        p4168582468: Chiller_3.Oil_temp_receiver
    Label (730,633 179x22), "Oil temperature receiver"
    Textfield (780,605 78x25), "%1.2f bar", text variable: Chiller_3.Oil_diff_pressure
        p4168582468: Chiller_3.Oil_diff_pressure
    Label (752,584 133x22), "Oil diff pressure"
    Label (720,136 139x24), "Prerotary position"
    Textfield (744,159 72x25), "%1.0f %%", text variable: Chiller_3.Feedback_PRV
        p4168582468: Chiller_3.Feedback_PRV
    Label (1067,211 200x24), "Suction pressure saturated"
    Textfield (1116,234 72x25), "%1.1f °C", text variable: Chiller_3.Suction_saturated_temp
        p4168582468: Chiller_3.Suction_saturated_temp
    Textfield (1116,291 72x25), "%1.1f bara", text variable: Chiller_3.Press_suction_compr
        p4168582468: Chiller_3.Press_suction_compr
    Label (1067,268 200x24), "Suction pressure"
    Textfield (1116,368 72x25), "%1.1f °C", text variable: Chiller_3.Theta_out
        p4168582468: Chiller_3.Theta_out
    Label (1111,345 83x24), "Theta out"
    Label (1196,557 104x27), "CW pressure"
    Textfield (1200,581 77x25), "%1.2f bar", text variable: Chiller_3.Press_chilled_medium_out
        p4168582468: Chiller_3.Press_chilled_medium_out
    Textfield (1200,710 77x25), "%1.2f bar", text variable: Chiller_3.Press_chilled_medium_in
        p4168582468: Chiller_3.Press_chilled_medium_in
    Label (1196,686 108x27), "CW pressure"
    Textfield (1170,506 72x25), "%1.1f °C", text variable: Chiller_3.Temp_chilled_medium_out
        p4168582468: Chiller_3.Temp_chilled_medium_out
    Label (1133,483 154x24), "Chilled water outlet"
    Label (1146,428 121x24), "CW setpoint"
    Textfield (1170,451 72x25), "%1.1f °C", text variable: Chiller_3.SP_PID_compressor
        p4168582468: Chiller_3.SP_PID_compressor
    Label (1239,619 113x30), "Diff pressure"
    Textfield (1256,648 77x25), "%1.2f bar", text variable: Chiller_3.dP_CW
        p4168582468: Chiller_3.dP_CW
    Textfield (1170,783 72x25), "%1.1f °C", text variable: Chiller_3.Temp_chilled_medium_in
        p4168582468: Chiller_3.Temp_chilled_medium_in
    Label (1133,760 148x24), "Chilled water inlet"
    Group (6,271 190x25)
        Rectangle (0,0 190x25)
        Label (0,2 105x21), "Running"
        Lamp1 (166,3 23x20), variable: Chiller_3.Unit_running, style: Lamp-Lamp1-Green
    Group (6,163 190x25)
        Rectangle (0,0 190x25)
        Label (1,2 105x21), "Auto"
        Lamp1 (166,3 23x20), variable: Chiller_3.Unit_auto, style: Lamp-Lamp1-Green
    Group (6,199 190x25)
        Rectangle (0,0 190x25)
        Label (0,2 105x21), "Remote"
        Lamp1 (166,3 23x20), variable: Chiller_3.Unit_remote, style: Lamp-Lamp1-Green
    Group (6,235 190x25)
        Rectangle (0,0 190x25)
        Label (0,2 105x21), "Manual"
        Lamp1 (166,3 23x20), variable: Chiller_3.Unit_manual, style: Lamp-Lamp1-Green
    Group (6,307 190x25)
        Rectangle (0,0 190x25)
        Label (1,2 105x21), "Available"
        Lamp1 (166,3 23x20), variable: Chiller_3.Unit_available, style: Lamp-Lamp1-Green
    Group (6,343 190x25)
        Rectangle (0,0 190x25)
        Label (0,2 130x21), "Start switch"
        Lamp1 (166,3 23x20), variable: Chiller_3.Unit_start_switch, style: Lamp-Lamp1-Green
    Group (6,381 190x25)
        Rectangle (0,0 190x25)
        Label (0,2 160x21), "Comms sequence"
        Lamp1 (166,3 23x20), variable: Sequence.A_Comms_Chiller_1, style: Lamp-Lamp1-Green
    Label (912,265 112x24), "Oil temp comp."
    Textfield (923,288 72x25), "%1.1f °C", text variable: Chiller_3.Temp_oil_inlet_compr
        p4168582468: Chiller_3.Temp_oil_inlet_compr
    Label (902,324 131x24), "Oil pressure [HP]"
    Textfield (923,347 72x25), "%1.2f bar", text variable: Chiller_3.Press_oil_compr
        p4168582468: Chiller_3.Press_oil_compr
    Image (921,41 317x130), invisible if: Chiller_3.Unit_alarm, image: ImagePool.ALARM
    Image (921,41 317x130), invisible if: Chiller_3.Unit_trip, image: ImagePool.TRIP
    Label (7,87 89x30), "Mode"
    Label (106,87 89x30), "Status"
    Rectangle (334,160 48x246)
    Image (238,160 48x246), image: ImagePool.CapBarTranparant
    BarDisplayImage (239,161 46x242), value: Sequence.Seq_cap_order_C1, style: BarDisplayImage-Gray, scale format: %.0f, scale 0..100
        p3451962224: ImagePool.Invisible
    Image (334,160 48x246), image: ImagePool.CapBarTranparant
    BarDisplayImage (335,161 46x242), value: Chiller_3.Chiller_capacity, style: BarDisplayImage-Gray, scale format: %.0f, scale 0..100
        p3451962224: ImagePool.Invisible
    Group (40,604 180x72)
        Rectangle (0,0 180x72)
        Label (0,0 180x72), "Sea water valve Pos. 100% = Max. overboard Pos. 0% = Max. recirculation"
    Rectangle (493,624 28x52)
    Image (493,624 29x54), image: ImagePool.CapBarTranparant
    BarDisplayImage (494,625 27x51), value: Chiller_3.Liquid_level_condenser, style: BarDisplayImage-Gray, scale format: %.0f, scale 0..100
        p3451962224: ImagePool.Invisible
    Rectangle (673,210 36x36), colour toggle: Chiller_3.Unit_running
    Rectangle (673,210 36x36), colour toggle: Chiller_3.Unit_alarm
    Rectangle (673,210 36x36), colour toggle: Chiller_3.Unit_trip
    Label (470,27 188x30), "Temp motor bearing"
    Textfield (525,84 77x25), "%1.1f °C", text variable: Chiller_3.Temp_motor_bearing_NDE
        p4168582468: Chiller_3.Temp_motor_bearing_NDE
    Textfield (525,54 77x25), "%1.1f °C", text variable: Chiller_3.Temp_motor_bearing_DE
        p4168582468: Chiller_3.Temp_motor_bearing_DE
    Label (480,54 37x25), "DE"
    Label (480,84 37x25), "NDE"
    Label (489,132 146x30), "Temp winding"
    Textfield (526,194 77x25), "%1.1f °C", text variable: Chiller_3.Temp_motor_wind_R
        p4168582468: Chiller_3.Temp_motor_wind_R
    Label (494,194 25x25), "R"
    Textfield (526,225 77x25), "%1.1f °C", text variable: Chiller_3.Temp_motor_wind_S
        p4168582468: Chiller_3.Temp_motor_wind_S
    Label (494,225 25x25), "S"
    Textfield (526,256 77x25), "%1.1f °C", text variable: Chiller_3.Temp_motor_wind_T
        p4168582468: Chiller_3.Temp_motor_wind_T
    Label (494,256 25x25), "T"
    Label (482,160 37x30), "Air"
    Textfield (526,163 77x25), "%1.1f °C", text variable: Chiller_3.Temp_motor_air
        p4168582468: Chiller_3.Temp_motor_air
    Textfield (411,508 76x25), "%1.1f °C", text variable: Chiller_3.Temp_water_outlet_cond
        p4168582468: Chiller_3.Temp_water_outlet_cond
    Label (390,478 127x30), "Sea water outlet"
    Label (720,86 139x24), "VGD Position"
    Textfield (744,109 72x25), "%1.0f %%", tooltip "Chiller_3.Feedback_VGD", text variable: Chiller_3.Feedback_VGD
    Label (720,31 139x24), "Stall detector"
    Textfield (744,54 72x25), "%1.0f V", text variable: Chiller_3.Stall_detector
        p4168582468: Chiller_3.Feedback_PRV
END_VISUALIZATION

// /Chiller_3_Oil
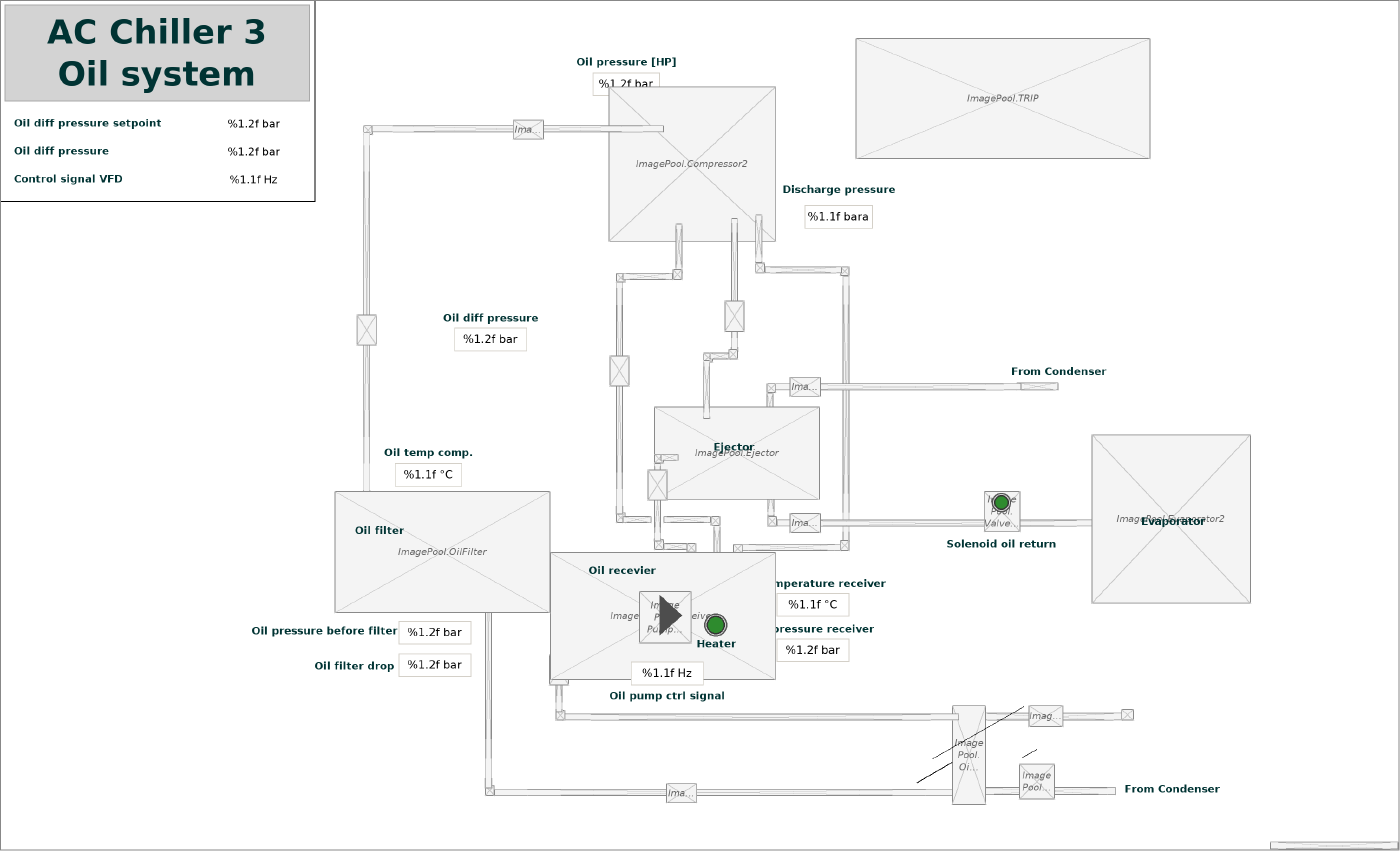
VISUALIZATION Chiller_3_Oil  // 1507x917
    Image (1094,412 45x8), angle 180, image: ImagePool.PipeBlack_1S_H_Faded
    Rectangle (0,0 339x217)
    Image (1367,907 138x8), angle 270, image: ImagePool.PipeGrey_1S_Horizontal
    Image (1053,768 155x8), image: ImagePool.PipeGrey_1S_Horizontal
    Image (1207,764 13x12), image: ImagePool.PipeGrey_3_LU
    Textfield (5,5 328x104), "AC Chiller 3 Oil system"
    Label (1066,387 128x27), "From Condenser"
    Label (838,191 129x27), "Discharge pressure"
    Textfield (866,221 73x25), "%1.1f bara", text variable: Chiller_3.Press_discharge_compr
        p4168582468: Chiller_3.Press_discharge_compr
    Label (1007,573 142x27), "Solenoid oil return"
    Textfield (429,704 78x25), "%1.2f bar", text variable: Chiller_3.Oil_Filter_Drop
        p4168582468: Chiller_3.Oil_Filter_Drop
    Label (340,707 83x22), "Oil filter drop"
    Textfield (836,688 78x25), "%1.2f bar", text variable: Chiller_3.Press_oil_receiver
        p4168582468: Chiller_3.Press_oil_receiver
    Label (808,667 135x22), "Oil pressure receiver"
    Textfield (836,639 78x25), "%1.1f °C", text variable: Chiller_3.Oil_temp_receiver
        p4168582468: Chiller_3.Oil_temp_receiver
    Label (804,618 143x22), "Oil temperature receiver"
    Textfield (489,353 78x25), "%1.2f bar", text variable: Chiller_3.Oil_diff_pressure
        p4168582468: Chiller_3.Oil_diff_pressure
    Label (478,332 101x22), "Oil diff pressure"
    Label (414,476 95x24), "Oil temp comp."
    Textfield (425,499 72x25), "%1.1f °C", text variable: Chiller_3.Temp_oil_inlet_compr
        p4168582468: Chiller_3.Temp_oil_inlet_compr
    Label (617,55 115x24), "Oil pressure [HP]"
    Textfield (638,78 72x25), "%1.2f bar", text variable: Chiller_3.Press_oil_compr
        p4168582468: Chiller_3.Press_oil_compr
    Image (921,41 317x130), invisible if: Chiller_3.Unit_alarm, image: ImagePool.ALARM
    Image (921,41 317x130), invisible if: Chiller_3.Unit_trip, image: ImagePool.TRIP
    Textfield (238,122 70x23), "%1.2f bar", text variable: Chiller_3.SP_oil_pressure
    Label (12,118 193x30), "Oil diff pressure setpoint"
    Textfield (238,152 70x23), "%1.2f bar", text variable: Chiller_3.Oil_diff_pressure
    Label (12,148 193x30), "Oil diff pressure"
    Textfield (238,182 70x23), "%1.1f Hz", text variable: Chiller_3.Setpoint_conv_oil_pump
    Label (12,178 131x30), "Control signal VFD"
    Label (651,739 135x22), "Oil pump ctrl signal"
    Textfield (429,669 78x25), "%1.2f bar", text variable: Chiller_3.Oil_pressure_before_filter
        p4168582468: Chiller_3.Oil_pressure_before_filter
    Label (276,669 147x22), "Oil pressure before filter"
    Label (1210,837 106x27), "From Condenser"
    Image (655,93 180x167), image: ImagePool.Compressor2
    Image (1051,848 150x8), angle 180, image: ImagePool.PipeBlack_1S_H_Faded
    Image (798,586 108x7), image: ImagePool.PipeBlack_1_Horizontal
    Image (907,297 7x286), image: ImagePool.PipeBlack_1_Vertical
    Image (391,135 10x10), image: ImagePool.PipeBlack_1_RD
    Image (522,846 10x11), image: ImagePool.PipeBlack_1_RU
    Image (1107,760 37x23), image: ImagePool.Arrow gray right
    Image (836,560 348x7), image: ImagePool.PipeBlack_1_Horizontal
    Image (1175,468 171x182), image: ImagePool.Evaporator2
    Image (826,512 7x44), image: ImagePool.PipeBlack_1_Vertical
    Image (826,556 10x11), image: ImagePool.PipeBlack_1_RU
    Image (789,596 7x28), image: ImagePool.PipeBlack_1_Vertical
    Image (789,586 10x10), image: ImagePool.PipeBlack_1_RD
    Image (904,582 10x11), image: ImagePool.PipeBlack_1_LU
    Image (850,553 33x21), image: ImagePool.Arrow black left
    Image (904,287 10x10), image: ImagePool.PipeBlack_1_LD
    Image (823,287 83x7), image: ImagePool.PipeBlack_1_Horizontal
    Image (813,283 10x11), image: ImagePool.PipeBlack_1_RU
    Image (813,231 7x52), image: ImagePool.PipeBlack_1_Vertical
    Image (825,413 10x10), image: ImagePool.PipeBlack_1_RD
    Image (834,413 265x7), image: ImagePool.PipeBlack_1_Horizontal
    Image (825,423 7x28), image: ImagePool.PipeBlack_1_Vertical
    Image (704,438 178x100), image: ImagePool.Ejector
    Image (850,406 33x21), image: ImagePool.Arrow black left
    Image (532,850 500x7), image: ImagePool.PipeBlack_1_Horizontal
    Image (1025,760 36x107), image: ImagePool.OilHeatExchanger
    Image (605,769 427x7), image: ImagePool.PipeBlack_1_Horizontal
    Image (598,765 10x11), image: ImagePool.PipeBlack_1_RU
    Image (598,670 7x97), image: ImagePool.PipeBlack_1_Vertical
    Image (598,660 10x10), image: ImagePool.PipeBlack_1_RD
    Image (605,660 19x7), image: ImagePool.PipeBlack_1_Horizontal
    Image (591,705 21x33), image: ImagePool.Arrow black down
    Image (717,844 33x21), image: ImagePool.Arrow black left
    Image (768,566 7x50), image: ImagePool.PipeBlack_1_Vertical
    Image (765,556 10x10), image: ImagePool.PipeBlack_1_LD
    Image (714,556 51x7), image: ImagePool.PipeBlack_1_Horizontal
    Image (704,581 10x11), image: ImagePool.PipeBlack_1_RU
    Image (704,499 7x84), image: ImagePool.PipeBlack_1_Vertical
    Image (704,489 10x10), image: ImagePool.PipeBlack_1_RD
    Image (711,489 19x7), image: ImagePool.PipeBlack_1_Horizontal
    Image (697,506 21x33), image: ImagePool.Arrow black down
    Image (714,585 28x7), image: ImagePool.PipeBlack_1_Horizontal
    Image (739,585 10x10), image: ImagePool.PipeBlack_1_LD
    Image (742,595 7x21), image: ImagePool.PipeBlack_1_Vertical
    Image (592,595 243x137), image: ImagePool.OilReceiver
    Image (400,135 314x7), image: ImagePool.PipeBlack_1_Horizontal
    Label (630,604 80x22), "Oil recevier"
    Image (522,553 7x296), image: ImagePool.PipeBlack_1_Vertical
    Image (519,544 10x10), image: ImagePool.PipeBlack_1_LD
    Image (400,544 120x7), image: ImagePool.PipeBlack_1_Horizontal
    Image (391,540 10x11), image: ImagePool.PipeBlack_1_RU
    Image (391,142 7x400), image: ImagePool.PipeBlack_1_Vertical
    Image (663,552 10x11), image: ImagePool.PipeBlack_1_RU
    Image (663,301 7x253), image: ImagePool.PipeBlack_1_Vertical
    Image (663,294 10x10), image: ImagePool.PipeBlack_1_RD
    Image (670,294 54x7), image: ImagePool.PipeBlack_1_Horizontal
    Image (656,383 21x33), image: ImagePool.Arrow black down
    Image (670,556 31x7), image: ImagePool.PipeBlack_1_Horizontal
    Image (727,241 7x53), image: ImagePool.PipeBlack_1_Vertical
    Image (724,290 10x11), image: ImagePool.PipeBlack_1_LU
    Image (757,380 10x10), image: ImagePool.PipeBlack_1_RD
    Image (764,380 22x7), image: ImagePool.PipeBlack_1_Horizontal
    Image (787,235 7x144), image: ImagePool.PipeBlack_1_Vertical
    Image (784,376 10x11), image: ImagePool.PipeBlack_1_LU
    Image (757,388 7x63), image: ImagePool.PipeBlack_1_Vertical
    Image (780,324 21x33), image: ImagePool.Arrow black down
    Label (750,471 80x22), "Ejector"
    Label (1223,551 80x22), "Evaporator"
    Image (384,339 21x33), image: ImagePool.Arrow black up
    Image (552,129 33x21), image: ImagePool.Arrow black right
    Image (360,529 232x131), image: ImagePool.OilFilter
    Label (379,561 59x22), "Oil filter"
    Line (987,843) (1025,821)
    Line (1100,816) (1116,807)
    Line (1004,817) (1102,761)
    Image (1097,823 38x38), image: ImagePool.RegValve
    Image (688,637 56x56), image: ImagePool.Pump_Large_3
    Polygon (710,660) (710,641) (734,663) (710,684) (710,676), colour toggle: Chiller_3.Comp_oil_pump
    Lamp1 (756,656 29x35), variable: Chiller_3.Oil_heater, style: Lamp-Lamp1-Green
    Label (744,683 55x22), "Heater"
    Image (1059,529 39x44), image: ImagePool.Valve_2
    Lamp1 (1066,529 24x25), variable: Chiller_3.Solenoid_oil_return, style: Lamp-Lamp1-Green
    Textfield (679,713 78x25), "%1.1f Hz", text variable: Chiller_3.Setpoint_conv_oil_pump
END_VISUALIZATION

// /Chiller_3_Trip
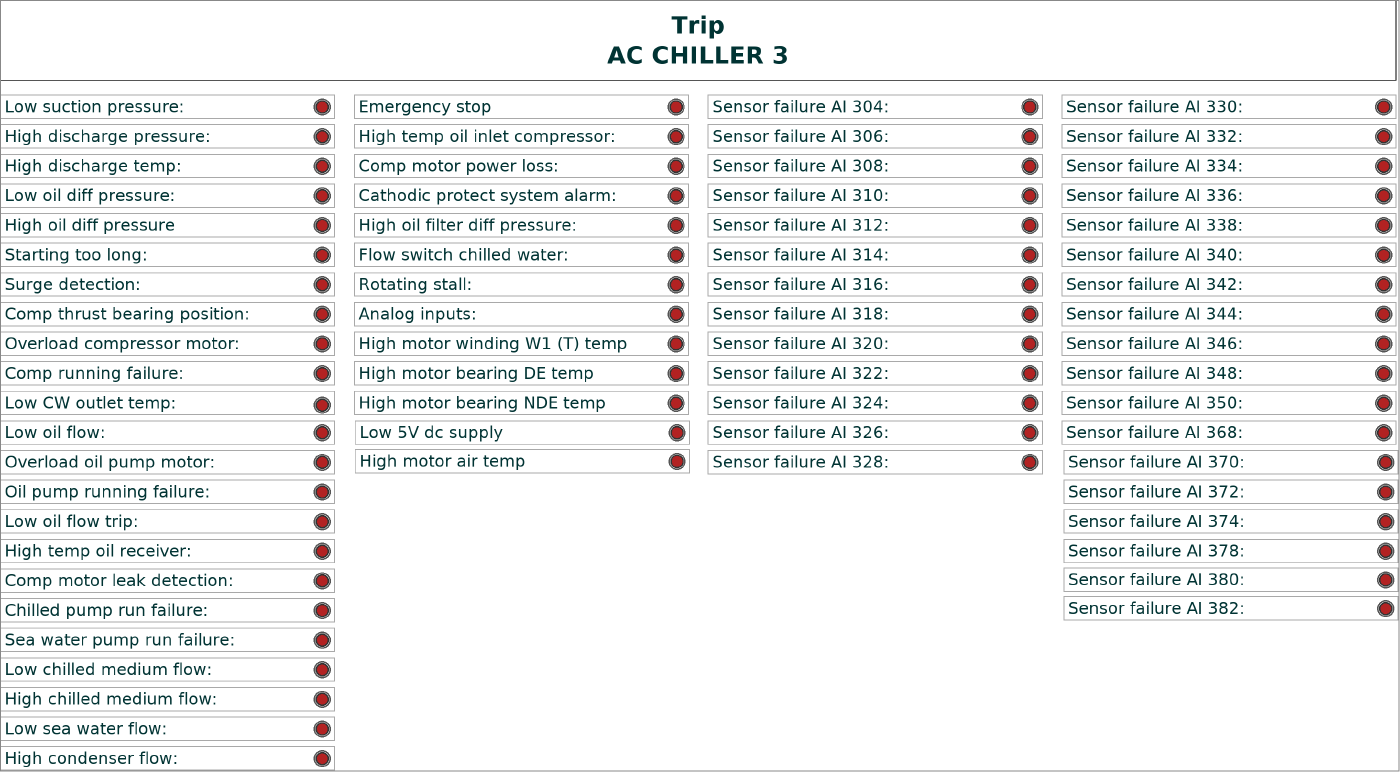
VISUALIZATION Chiller_3_Trip  // 1464x808
    Rectangle (0,0 1460x84)
    Label (274,7 912x70), "Trip AC CHILLER 3"
    Group (0,99 350x25)
        Rectangle (0,0 350x25)
        Label (2,2 319x21), "Low suction pressure:"
        Lamp1 (326,3 22x20), variable: not.Chiller_3.T_Low_suction_pressure, style: Lamp-Lamp1-Red
    Group (0,130 350x25)
        Rectangle (0,0 350x25)
        Label (2,2 319x21), "High discharge pressure:"
        Lamp1 (326,3 22x20), variable: not.Chiller_3.T_High_discharge_pressure, style: Lamp-Lamp1-Red
    Group (0,161 350x25)
        Rectangle (0,0 350x25)
        Label (2,2 319x21), "High discharge temp:"
        Lamp1 (326,3 22x20), variable: not.Chiller_3.T_High_discharge_temp, style: Lamp-Lamp1-Red
    Group (0,192 350x25)
        Rectangle (0,0 350x25)
        Label (2,2 319x21), "Low oil diff pressure:"
        Lamp1 (326,3 22x20), variable: not.Chiller_3.T_Low_oil_diff_pressure, style: Lamp-Lamp1-Red
    Group (0,223 350x25)
        Rectangle (0,0 350x25)
        Label (2,2 319x21), "High oil diff pressure"
        Lamp1 (326,3 22x20), variable: not.Chiller_3.T_High_diff_oil_pressure, style: Lamp-Lamp1-Red
    Group (0,254 350x25)
        Rectangle (0,0 350x25)
        Label (2,2 319x21), "Starting too long:"
        Lamp1 (326,3 22x20), variable: not.Chiller_3.T_Starting_to_long, style: Lamp-Lamp1-Red
    Group (0,285 350x25)
        Rectangle (0,0 350x25)
        Label (2,2 319x21), "Surge detection:"
        Lamp1 (326,3 22x20), variable: not.Chiller_3.T_Surge_detection, style: Lamp-Lamp1-Red
    Group (0,316 350x25)
        Rectangle (0,0 350x25)
        Label (2,2 319x21), "Comp thrust bearing position:"
        Lamp1 (326,3 22x20), variable: not.Chiller_3.T_Comp_thrust_bearing_position, style: Lamp-Lamp1-Red
    Group (0,347 350x25)
        Rectangle (0,0 350x25)
        Label (2,2 319x21), "Overload compressor motor:"
        Lamp1 (326,3 22x20), variable: not.Chiller_3.T_Overload_compressor_motor, style: Lamp-Lamp1-Red
    Group (0,378 350x25)
        Rectangle (0,0 350x25)
        Label (2,2 319x21), "Comp running failure:"
        Lamp1 (326,3 22x20), variable: not.Chiller_3.T_Compressor_running_failure, style: Lamp-Lamp1-Red
    Group (0,440 350x25)
        Rectangle (0,0 350x25)
        Label (2,2 319x21), "Low oil flow:"
        Lamp1 (326,3 22x20), variable: not.Chiller_3.T_Low_oil_flow, style: Lamp-Lamp1-Red
    Group (0,471 350x25)
        Rectangle (0,0 350x25)
        Label (2,2 319x21), "Overload oil pump motor:"
        Lamp1 (326,3 22x20), variable: not.Chiller_3.T_Overload_oil_pump_motor, style: Lamp-Lamp1-Red
    Group (0,502 350x25)
        Rectangle (0,0 350x25)
        Label (2,2 319x21), "Oil pump running failure:"
        Lamp1 (326,3 22x20), variable: not.Chiller_3.T_Oil_pump_running_failure, style: Lamp-Lamp1-Red
    Group (0,533 350x25)
        Rectangle (0,0 350x25)
        Label (2,2 319x21), "Low oil flow trip:"
        Lamp1 (326,3 22x20), variable: not.Chiller_3.T_Low_oil_flow_trip, style: Lamp-Lamp1-Red
    Group (0,564 350x25)
        Rectangle (0,0 350x25)
        Label (2,2 319x21), "High temp oil receiver:"
        Lamp1 (326,3 22x20), variable: not.Chiller_3.T_High_temp_oil_receiver, style: Lamp-Lamp1-Red
    Group (0,595 350x25)
        Rectangle (0,0 350x25)
        Label (2,2 319x21), "Comp motor leak detection:"
        Lamp1 (326,3 22x20), variable: not.Chiller_3.T_Comp_motor_leak_detection, style: Lamp-Lamp1-Red
    Group (0,626 350x25)
        Rectangle (0,0 350x25)
        Label (2,2 319x21), "Chilled pump run failure:"
        Lamp1 (326,3 22x20), variable: not.Chiller_3.T_Chilled_pump_run_failure, style: Lamp-Lamp1-Red
    Rectangle (0,688 350x25)
    Label (2,690 319x21), "Low chilled medium flow:"
    Lamp1 (326,691 22x20), variable: not.Chiller_3.T_Low_chilled_medium_flow, style: Lamp-Lamp1-Red
    Group (0,657 350x25)
        Rectangle (0,0 350x25)
        Label (2,2 319x21), "Sea water pump run failure:"
        Lamp1 (326,3 22x20), variable: not.Chiller_3.T_Sea_water_pump_run_failure, style: Lamp-Lamp1-Red
    Rectangle (0,719 350x25)
    Label (2,721 319x21), "High chilled medium flow:"
    Lamp1 (326,722 22x20), variable: not.Chiller_3.T_High_chilled_medium_flow, style: Lamp-Lamp1-Red
    Rectangle (0,750 350x25)
    Label (2,752 319x21), "Low sea water flow:"
    Lamp1 (326,753 22x20), variable: not.Chiller_3.T_Low_sea_water_flow, style: Lamp-Lamp1-Red
    Group (0,781 350x25)
        Rectangle (0,0 350x25)
        Label (2,2 319x21), "High condenser flow:"
        Lamp1 (326,3 22x20), variable: not.Chiller_3.T_High_condenser_flow, style: Lamp-Lamp1-Red
    Group (1110,99 350x25)
        Rectangle (0,0 350x25)
        Label (2,2 319x21), "Sensor failure AI 330:"
        Lamp1 (326,3 22x20), variable: not.Chiller_3.T_Sensor_failure_AI_330, style: Lamp-Lamp1-Red
    Group (1110,130 350x25)
        Rectangle (0,0 350x25)
        Label (2,2 319x21), "Sensor failure AI 332:"
        Lamp1 (326,3 22x20), variable: not.Chiller_3.T_Sensor_failure_AI_332, style: Lamp-Lamp1-Red
    Group (1110,161 350x25)
        Rectangle (0,0 350x25)
        Label (2,2 319x21), "Sensor failure AI 334:"
        Lamp1 (326,3 22x20), variable: not.Chiller_3.T_Sensor_failure_AI_334, style: Lamp-Lamp1-Red
    Group (740,223 350x25)
        Rectangle (0,0 350x25)
        Label (2,2 319x21), "Sensor failure AI 312:"
        Lamp1 (326,3 22x20), variable: not.Chiller_3.T_Sensor_failure_AI_312, style: Lamp-Lamp1-Red
    Group (740,254 350x25)
        Rectangle (0,0 350x25)
        Label (2,2 319x21), "Sensor failure AI 314:"
        Lamp1 (326,3 22x20), variable: not.Chiller_3.T_Sensor_failure_AI_314, style: Lamp-Lamp1-Red
    Group (740,285 350x25)
        Rectangle (0,0 350x25)
        Label (2,2 319x21), "Sensor failure AI 316:"
        Lamp1 (326,3 22x20), variable: not.Chiller_3.T_Sensor_failure_AI_316, style: Lamp-Lamp1-Red
    Group (740,316 350x25)
        Rectangle (0,0 350x25)
        Label (2,2 319x21), "Sensor failure AI 318:"
        Lamp1 (326,3 22x20), variable: not.Chiller_3.T_Sensor_failure_AI_318, style: Lamp-Lamp1-Red
    Group (1110,192 350x25)
        Rectangle (0,0 350x25)
        Label (2,2 319x21), "Sensor failure AI 336:"
        Lamp1 (326,3 22x20), variable: not.Chiller_3.T_Sensor_failure_AI_336, style: Lamp-Lamp1-Red
    Group (1110,223 350x25)
        Rectangle (0,0 350x25)
        Label (2,2 319x21), "Sensor failure AI 338:"
        Lamp1 (326,3 22x20), variable: not.Chiller_3.T_Sensor_failure_AI_338, style: Lamp-Lamp1-Red
    Rectangle (1110,409 350x25)
    Label (1112,411 319x21), "Sensor failure AI 350:"
    Lamp1 (1436,412 22x20), variable: not.Chiller_3.T_Sensor_failure_AI_350, style: Lamp-Lamp1-Red
    Group (1110,254 350x25)
        Rectangle (0,0 350x25)
        Label (2,2 319x21), "Sensor failure AI 340:"
        Lamp1 (326,3 22x20), variable: not.Chiller_3.T_Sensor_failure_AI_340, style: Lamp-Lamp1-Red
    Group (1110,285 350x25)
        Rectangle (0,0 350x25)
        Label (2,2 319x21), "Sensor failure AI 342:"
        Lamp1 (326,3 22x20), variable: not.Chiller_3.T_Sensor_failure_AI_342, style: Lamp-Lamp1-Red
    Rectangle (1110,316 350x25)
    Label (1112,318 319x21), "Sensor failure AI 344:"
    Lamp1 (1436,319 22x20), variable: not.Chiller_3.T_Sensor_failure_AI_344, style: Lamp-Lamp1-Red
    Group (1110,347 350x25)
        Rectangle (0,0 350x25)
        Label (2,2 319x21), "Sensor failure AI 346:"
        Lamp1 (326,3 22x20), variable: not.Chiller_3.T_Sensor_failure_AI_346, style: Lamp-Lamp1-Red
    Rectangle (1110,378 350x25)
    Label (1112,380 319x21), "Sensor failure AI 348:"
    Lamp1 (1436,381 22x20), variable: not.Chiller_3.T_Sensor_failure_AI_348, style: Lamp-Lamp1-Red
    Group (1110,440 350x25)
        Rectangle (0,0 350x25)
        Label (2,2 319x21), "Sensor failure AI 368:"
        Lamp1 (326,3 22x20), variable: not.Chiller_3.T_Sensor_failure_AI_368, style: Lamp-Lamp1-Red
    Group (740,378 350x25)
        Rectangle (0,0 350x25)
        Label (2,2 319x21), "Sensor failure AI 322:"
        Lamp1 (326,3 22x20), variable: not.Chiller_3.T_Sensor_failure_AI_322, style: Lamp-Lamp1-Red
    Group (740,409 350x25)
        Rectangle (0,0 350x25)
        Label (2,2 319x21), "Sensor failure AI 324:"
        Lamp1 (326,3 22x20), variable: not.Chiller_3.T_Sensor_failure_AI_324, style: Lamp-Lamp1-Red
    Group (740,440 350x25)
        Rectangle (0,0 350x25)
        Label (2,2 319x21), "Sensor failure AI 326:"
        Lamp1 (326,3 22x20), variable: not.Chiller_3.T_Sensor_failure_AI_326, style: Lamp-Lamp1-Red
    Group (740,471 350x25)
        Rectangle (0,0 350x25)
        Label (2,2 319x21), "Sensor failure AI 328:"
        Lamp1 (326,3 22x20), variable: not.Chiller_3.T_Sensor_failure_AI_328, style: Lamp-Lamp1-Red
    Group (1112,502 350x25)
        Rectangle (0,0 350x25)
        Label (2,2 319x21), "Sensor failure AI 372:"
        Lamp1 (326,3 22x20), variable: not.Chiller_3.T_Sensor_failure_AI_372, style: Lamp-Lamp1-Red
    Group (1112,533 350x25)
        Rectangle (0,0 350x25)
        Label (2,2 319x21), "Sensor failure AI 374:"
        Lamp1 (326,3 22x20), variable: not.Chiller_3.T_Sensor_failure_AI_374, style: Lamp-Lamp1-Red
    Group (1112,564 350x25)
        Rectangle (0,0 350x25)
        Label (2,2 319x21), "Sensor failure AI 378:"
        Lamp1 (326,3 22x20), variable: not.Chiller_3.T_Sensor_failure_AI_378, style: Lamp-Lamp1-Red
    Group (740,347 350x25)
        Rectangle (0,0 350x25)
        Label (2,2 319x21), "Sensor failure AI 320:"
        Lamp1 (326,3 22x20), variable: not.Chiller_3.T_Sensor_failure_AI_320, style: Lamp-Lamp1-Red
    Group (740,99 350x25)
        Rectangle (0,0 350x25)
        Label (2,2 319x21), "Sensor failure AI 304:"
        Lamp1 (326,3 22x20), variable: not.Chiller_3.T_Sensor_failure_AI_304, style: Lamp-Lamp1-Red
    Group (740,130 350x25)
        Rectangle (0,0 350x25)
        Label (2,2 319x21), "Sensor failure AI 306:"
        Lamp1 (326,3 22x20), variable: not.Chiller_3.T_Sensor_failure_AI_306, style: Lamp-Lamp1-Red
    Group (740,161 350x25)
        Rectangle (0,0 350x25)
        Label (2,2 319x21), "Sensor failure AI 308:"
        Lamp1 (326,3 22x20), variable: not.Chiller_3.T_Sensor_failure_AI_308, style: Lamp-Lamp1-Red
    Group (740,192 350x25)
        Rectangle (0,0 350x25)
        Label (2,2 319x21), "Sensor failure AI 310:"
        Lamp1 (326,3 22x20), variable: not.Chiller_3.T_Sensor_failure_AI_310, style: Lamp-Lamp1-Red
    Rectangle (1112,471 350x25)
    Label (1114,473 319x21), "Sensor failure AI 370:"
    Lamp1 (1438,474 22x20), variable: not.Chiller_3.T_Sensor_failure_AI_370, style: Lamp-Lamp1-Red
    Group (370,99 350x25)
        Rectangle (0,0 350x25)
        Label (2,2 319x21), "Emergency stop"
        Lamp1 (326,3 22x20), variable: not.Chiller_3.T_Emergency_stop, style: Lamp-Lamp1-Red
    Group (370,130 350x25)
        Rectangle (0,0 350x25)
        Label (2,2 319x21), "High temp oil inlet compressor:"
        Lamp1 (326,3 22x20), variable: not.Chiller_3.T_High_temp_oil_inlet_comp, style: Lamp-Lamp1-Red
    Group (370,161 350x25)
        Rectangle (0,0 350x25)
        Label (2,2 319x21), "Comp motor power loss:"
        Lamp1 (326,3 22x20), variable: not.Chiller_3.T_Comp_motor_power_loss, style: Lamp-Lamp1-Red
    Group (370,192 350x25)
        Rectangle (0,0 350x25)
        Label (2,2 319x21), "Cathodic protect system alarm:"
        Lamp1 (326,3 22x20), variable: not.Chiller_3.T_Cathodic_protect_sys_alarm, style: Lamp-Lamp1-Red
    Group (370,223 350x25)
        Rectangle (0,0 350x25)
        Label (2,2 319x21), "High oil filter diff pressure:"
        Lamp1 (326,3 22x20), variable: not.Chiller_3.T_High_oil_filter_diff_press, style: Lamp-Lamp1-Red
    Rectangle (370,316 350x25)
    Label (372,318 319x21), "Analog inputs:"
    Lamp1 (696,319 22x20), variable: not.Chiller_3.T_Analog_inputs, style: Lamp-Lamp1-Red
    Group (370,254 350x25)
        Rectangle (0,0 350x25)
        Label (2,2 319x21), "Flow switch chilled water:"
        Lamp1 (326,3 22x20), variable: not.Chiller_3.T_Flow_switch_FT01, style: Lamp-Lamp1-Red
    Group (370,285 350x25)
        Rectangle (0,0 350x25)
        Label (2,2 319x21), "Rotating stall:"
        Lamp1 (326,3 22x20), variable: not.Chiller_3.T_Rotating_stall_trip, style: Lamp-Lamp1-Red
    Rectangle (0,409 350x25)
    Label (2,411 319x21), "Low CW outlet temp:"
    Group (1112,594 350x25)
        Rectangle (0,0 350x25)
        Label (2,2 319x21), "Sensor failure AI 380:"
        Lamp1 (326,3 22x20), variable: not.Chiller_3.T_Sensor_failure_AI_380, style: Lamp-Lamp1-Red
    Lamp1 (326,414 22x20), variable: not.Chiller_3.T_Low_chilled_medium_outlet, style: Lamp-Lamp1-Red
    Rectangle (370,347 350x25)
    Label (372,349 319x21), "High motor winding W1 (T) temp"
    Lamp1 (696,350 22x20), variable: not.Chiller_3.T_High_comp_motor_wind_temp, style: Lamp-Lamp1-Red
    Rectangle (370,378 350x25)
    Label (372,380 319x21), "High motor bearing DE temp"
    Lamp1 (696,381 22x20), variable: not.Chiller_3.T_High_comp_mot_DE_bear_temp, style: Lamp-Lamp1-Red
    Rectangle (370,409 350x25)
    Label (372,411 319x21), "High motor bearing NDE temp"
    Lamp1 (696,412 22x20), variable: not.Chiller_3.T_High_comp_mot_NDE_bear_temp, style: Lamp-Lamp1-Red
    Group (1112,624 350x25)
        Rectangle (0,0 350x25)
        Label (2,2 319x21), "Sensor failure AI 382:"
        Lamp1 (326,3 22x20), variable: not.Chiller_3.T_Sensor_failure_AI_382, style: Lamp-Lamp1-Red
    Rectangle (371,440 350x25)
    Label (373,442 319x21), "Low 5V dc supply"
    Lamp1 (697,443 22x20), variable: not.Chiller_3.T_Low_5VDC_supply, style: Lamp-Lamp1-Red
    Rectangle (371,470 350x25)
    Label (373,472 319x21), "High motor air temp"
    Lamp1 (697,473 22x20), variable: not.Chiller_3.T_High_motor_air_temp, style: Lamp-Lamp1-Red
END_VISUALIZATION

// /Chiller_4_Alarm
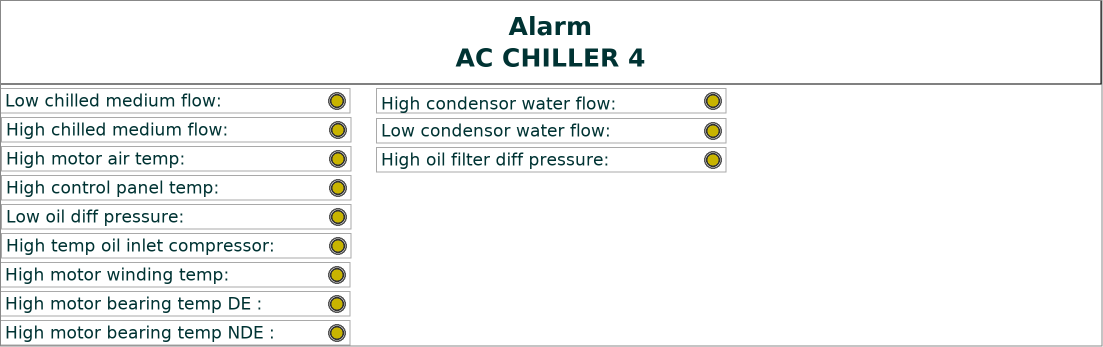
VISUALIZATION Chiller_4_Alarm  // 1103x347
    Rectangle (0,0 1101x84)
    Label (19,7 1063x70), "Alarm AC CHILLER 4"
    Rectangle (1,117 350x25)
    Label (3,119 314x21), "High chilled medium flow:"
    Lamp1 (327,120 22x20), variable: not.Chiller_4.A_High_chilled_medium_flow, style: Lamp-Lamp1-Yellow
    Rectangle (0,262 350x25)
    Label (2,264 314x21), "High motor winding temp:"
    Lamp1 (326,265 22x20), variable: not.Chiller_4.A_High_comp_motor_winding_temp, style: Lamp-Lamp1-Yellow
    Rectangle (0,291 350x25)
    Label (2,293 315x21), "High motor bearing temp DE :"
    Lamp1 (326,294 22x20), variable: not.Chiller_4.A_High_comp_mo_DE_bear_temp, style: Lamp-Lamp1-Yellow
    Rectangle (1,233 350x25)
    Label (3,235 312x21), "High temp oil inlet compressor:"
    Lamp1 (327,236 22x20), variable: not.Chiller_4.A_High_temp_oil_inlet_comp, style: Lamp-Lamp1-Yellow
    Rectangle (1,175 350x25)
    Label (3,177 309x21), "High control panel temp:"
    Lamp1 (327,178 22x20), variable: not.Chiller_4.A_High_control_panel_temp, style: Lamp-Lamp1-Yellow
    Rectangle (1,204 350x25)
    Label (3,206 315x21), "Low oil diff pressure:"
    Lamp1 (327,207 22x20), variable: not.Chiller_4.A_Low_oil_diff_pressure, style: Lamp-Lamp1-Yellow
    Rectangle (376,118 350x25)
    Label (378,120 320x21), "Low condensor water flow:"
    Lamp1 (702,121 22x20), variable: not.Chiller_4.A_Low_sea_water_flow, style: Lamp-Lamp1-Yellow
    Rectangle (376,147 350x25)
    Label (378,149 319x21), "High oil filter diff pressure:"
    Lamp1 (702,150 22x20), variable: not.Chiller_4.A_High_oil_filter_diff_press, style: Lamp-Lamp1-Yellow
    Rectangle (1,146 350x25)
    Label (3,148 314x21), "High motor air temp:"
    Lamp1 (327,149 22x20), variable: not.Chiller_4.A_High_motor_air_temp, style: Lamp-Lamp1-Yellow
    Rectangle (0,320 350x25)
    Label (2,322 315x21), "High motor bearing temp NDE :"
    Lamp1 (326,323 22x20), variable: not.Chiller_4.A_High_comp_mo_NDE_bear_temp, style: Lamp-Lamp1-Yellow
    Rectangle (0,88 350x25)
    Label (2,90 314x21), "Low chilled medium flow:"
    Lamp1 (326,91 22x20), variable: not.Chiller_4.A_Low_chilled_medium_flow, style: Lamp-Lamp1-Yellow
    Rectangle (376,88 350x25)
    Label (378,96 319x15), "High condensor water flow:"
    Lamp1 (702,91 22x20), variable: not.Chiller_4.A_High_condenser_flow, style: Lamp-Lamp1-Yellow
END_VISUALIZATION

// /Chiller_4_Alarm
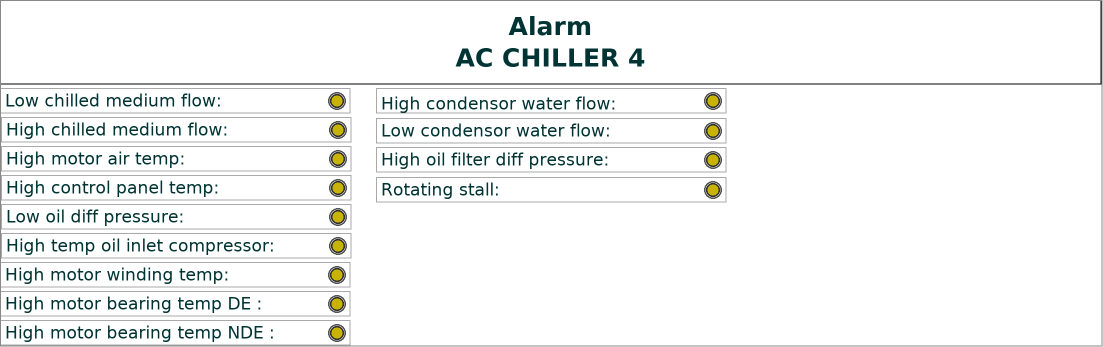
VISUALIZATION Chiller_4_Alarm  // 1103x347
    Rectangle (0,0 1101x84)
    Label (19,7 1063x70), "Alarm AC CHILLER 4"
    Rectangle (1,117 350x25)
    Label (3,119 314x21), "High chilled medium flow:"
    Lamp1 (327,120 22x20), variable: not.Chiller_4.A_High_chilled_medium_flow, style: Lamp-Lamp1-Yellow
    Rectangle (0,262 350x25)
    Label (2,264 314x21), "High motor winding temp:"
    Lamp1 (326,265 22x20), variable: not.Chiller_4.A_High_comp_motor_winding_temp, style: Lamp-Lamp1-Yellow
    Rectangle (0,291 350x25)
    Label (2,293 315x21), "High motor bearing temp DE :"
    Lamp1 (326,294 22x20), variable: not.Chiller_4.A_High_comp_mo_DE_bear_temp, style: Lamp-Lamp1-Yellow
    Rectangle (1,233 350x25)
    Label (3,235 312x21), "High temp oil inlet compressor:"
    Lamp1 (327,236 22x20), variable: not.Chiller_4.A_High_temp_oil_inlet_comp, style: Lamp-Lamp1-Yellow
    Rectangle (1,175 350x25)
    Label (3,177 309x21), "High control panel temp:"
    Lamp1 (327,178 22x20), variable: not.Chiller_4.A_High_control_panel_temp, style: Lamp-Lamp1-Yellow
    Rectangle (1,204 350x25)
    Label (3,206 315x21), "Low oil diff pressure:"
    Lamp1 (327,207 22x20), variable: not.Chiller_4.A_Low_oil_diff_pressure, style: Lamp-Lamp1-Yellow
    Rectangle (376,118 350x25)
    Label (378,120 320x21), "Low condensor water flow:"
    Lamp1 (702,121 22x20), variable: not.Chiller_4.A_Low_sea_water_flow, style: Lamp-Lamp1-Yellow
    Rectangle (376,147 350x25)
    Label (378,149 319x21), "High oil filter diff pressure:"
    Lamp1 (702,150 22x20), variable: not.Chiller_4.A_High_oil_filter_diff_press, style: Lamp-Lamp1-Yellow
    Rectangle (1,146 350x25)
    Label (3,148 314x21), "High motor air temp:"
    Lamp1 (327,149 22x20), variable: not.Chiller_4.A_High_motor_air_temp, style: Lamp-Lamp1-Yellow
    Rectangle (0,320 350x25)
    Label (2,322 315x21), "High motor bearing temp NDE :"
    Lamp1 (326,323 22x20), variable: not.Chiller_4.A_High_comp_mo_NDE_bear_temp, style: Lamp-Lamp1-Yellow
    Rectangle (0,88 350x25)
    Label (2,90 314x21), "Low chilled medium flow:"
    Lamp1 (326,91 22x20), variable: not.Chiller_4.A_Low_chilled_medium_flow, style: Lamp-Lamp1-Yellow
    Rectangle (376,88 350x25)
    Label (378,96 319x15), "High condensor water flow:"
    Lamp1 (702,91 22x20), variable: not.Chiller_4.A_High_condenser_flow, style: Lamp-Lamp1-Yellow
    Rectangle (376,177 350x25)
    Label (378,179 319x21), "Rotating stall:"
    Lamp1 (702,180 22x20), variable: not.Chiller_4.A_Rotating_stall, style: Lamp-Lamp1-Yellow
END_VISUALIZATION

// /Chiller_4_Oil
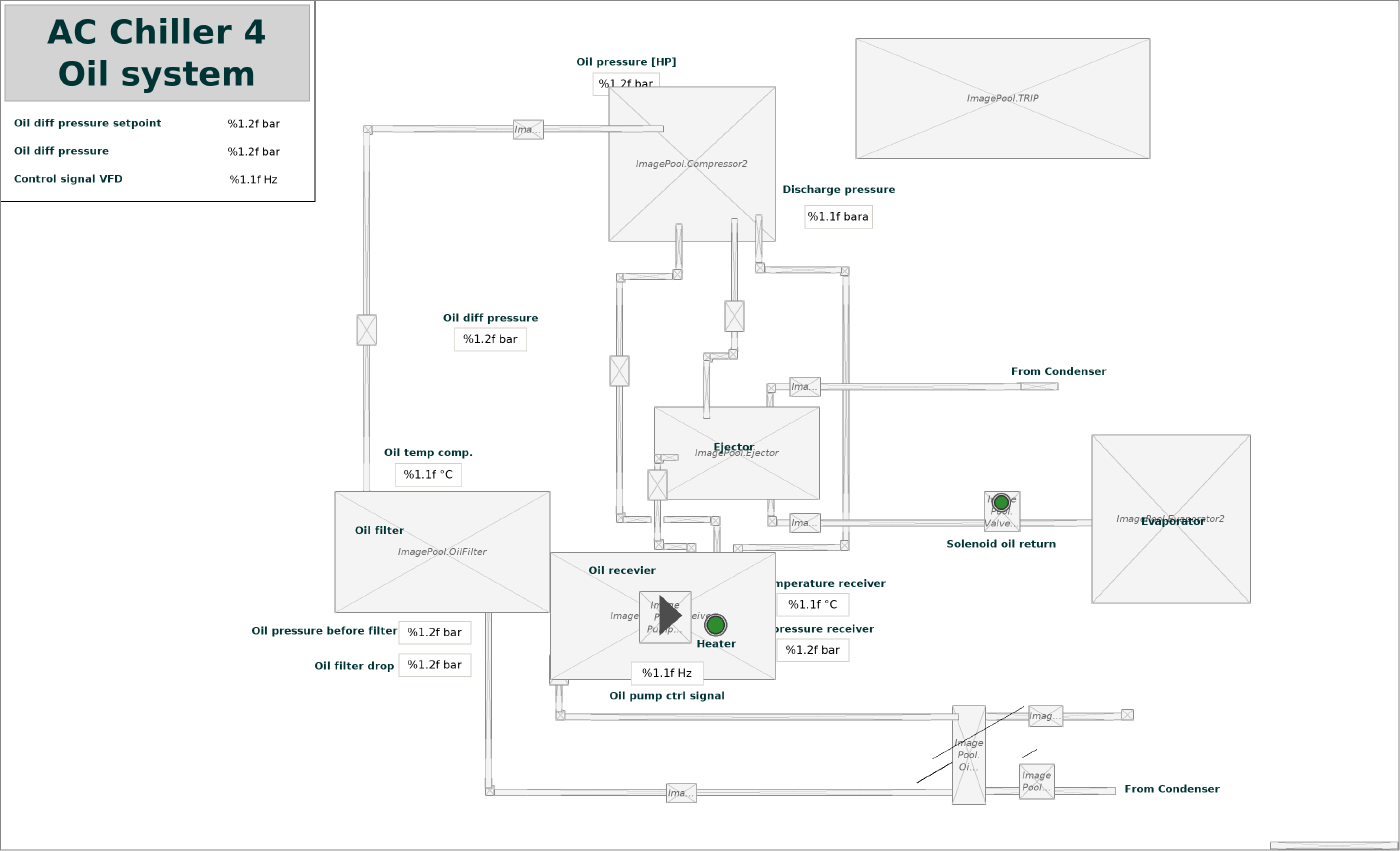
VISUALIZATION Chiller_4_Oil  // 1507x917
    Image (1094,412 45x8), angle 180, image: ImagePool.PipeBlack_1S_H_Faded
    Rectangle (0,0 339x217)
    Image (1367,907 138x8), angle 270, image: ImagePool.PipeGrey_1S_Horizontal
    Image (1053,768 155x8), image: ImagePool.PipeGrey_1S_Horizontal
    Image (1207,764 13x12), image: ImagePool.PipeGrey_3_LU
    Textfield (5,5 328x104), "AC Chiller 4 Oil system"
    Label (1066,387 128x27), "From Condenser"
    Label (838,191 129x27), "Discharge pressure"
    Textfield (866,221 73x25), "%1.1f bara", text variable: Chiller_4.Press_discharge_compr
        p4168582468: Chiller_4.Press_discharge_compr
    Label (1007,573 142x27), "Solenoid oil return"
    Textfield (429,704 78x25), "%1.2f bar", text variable: Chiller_4.Oil_Filter_Drop
        p4168582468: Chiller_4.Oil_Filter_Drop
    Label (340,707 83x22), "Oil filter drop"
    Textfield (836,688 78x25), "%1.2f bar", text variable: Chiller_4.Press_oil_receiver
        p4168582468: Chiller_4.Press_oil_receiver
    Label (808,667 135x22), "Oil pressure receiver"
    Textfield (836,639 78x25), "%1.1f °C", text variable: Chiller_4.Oil_temp_receiver
        p4168582468: Chiller_4.Oil_temp_receiver
    Label (804,618 143x22), "Oil temperature receiver"
    Textfield (489,353 78x25), "%1.2f bar", text variable: Chiller_4.Oil_diff_pressure
        p4168582468: Chiller_4.Oil_diff_pressure
    Label (478,332 101x22), "Oil diff pressure"
    Label (414,476 95x24), "Oil temp comp."
    Textfield (425,499 72x25), "%1.1f °C", text variable: Chiller_4.Temp_oil_inlet_compr
        p4168582468: Chiller_4.Temp_oil_inlet_compr
    Label (617,55 115x24), "Oil pressure [HP]"
    Textfield (638,78 72x25), "%1.2f bar", text variable: Chiller_4.Press_oil_compr
        p4168582468: Chiller_4.Press_oil_compr
    Image (921,41 317x130), invisible if: Chiller_4.Unit_alarm, image: ImagePool.ALARM
    Image (921,41 317x130), invisible if: Chiller_4.Unit_trip, image: ImagePool.TRIP
    Textfield (238,122 70x23), "%1.2f bar", text variable: Chiller_4.SP_oil_pressure
    Label (12,118 193x30), "Oil diff pressure setpoint"
    Textfield (238,152 70x23), "%1.2f bar", text variable: Chiller_4.Oil_diff_pressure
    Label (12,148 193x30), "Oil diff pressure"
    Textfield (238,182 70x23), "%1.1f Hz", text variable: Chiller_4.Setpoint_conv_oil_pump
    Label (12,178 131x30), "Control signal VFD"
    Label (651,739 135x22), "Oil pump ctrl signal"
    Textfield (429,669 78x25), "%1.2f bar", text variable: Chiller_4.Oil_pressure_before_filter
        p4168582468: Chiller_4.Oil_pressure_before_filter
    Label (276,669 147x22), "Oil pressure before filter"
    Label (1210,837 106x27), "From Condenser"
    Image (655,93 180x167), image: ImagePool.Compressor2
    Image (1051,848 150x8), angle 180, image: ImagePool.PipeBlack_1S_H_Faded
    Image (798,586 108x7), image: ImagePool.PipeBlack_1_Horizontal
    Image (907,297 7x286), image: ImagePool.PipeBlack_1_Vertical
    Image (391,135 10x10), image: ImagePool.PipeBlack_1_RD
    Image (522,846 10x11), image: ImagePool.PipeBlack_1_RU
    Image (1107,760 37x23), image: ImagePool.Arrow gray right
    Image (836,560 348x7), image: ImagePool.PipeBlack_1_Horizontal
    Image (1175,468 171x182), image: ImagePool.Evaporator2
    Image (826,512 7x44), image: ImagePool.PipeBlack_1_Vertical
    Image (826,556 10x11), image: ImagePool.PipeBlack_1_RU
    Image (789,596 7x28), image: ImagePool.PipeBlack_1_Vertical
    Image (789,586 10x10), image: ImagePool.PipeBlack_1_RD
    Image (904,582 10x11), image: ImagePool.PipeBlack_1_LU
    Image (850,553 33x21), image: ImagePool.Arrow black left
    Image (904,287 10x10), image: ImagePool.PipeBlack_1_LD
    Image (823,287 83x7), image: ImagePool.PipeBlack_1_Horizontal
    Image (813,283 10x11), image: ImagePool.PipeBlack_1_RU
    Image (813,231 7x52), image: ImagePool.PipeBlack_1_Vertical
    Image (825,413 10x10), image: ImagePool.PipeBlack_1_RD
    Image (834,413 265x7), image: ImagePool.PipeBlack_1_Horizontal
    Image (825,423 7x28), image: ImagePool.PipeBlack_1_Vertical
    Image (704,438 178x100), image: ImagePool.Ejector
    Image (850,406 33x21), image: ImagePool.Arrow black left
    Image (532,850 500x7), image: ImagePool.PipeBlack_1_Horizontal
    Image (1025,760 36x107), image: ImagePool.OilHeatExchanger
    Image (605,769 427x7), image: ImagePool.PipeBlack_1_Horizontal
    Image (598,765 10x11), image: ImagePool.PipeBlack_1_RU
    Image (598,670 7x97), image: ImagePool.PipeBlack_1_Vertical
    Image (598,660 10x10), image: ImagePool.PipeBlack_1_RD
    Image (605,660 19x7), image: ImagePool.PipeBlack_1_Horizontal
    Image (591,705 21x33), image: ImagePool.Arrow black down
    Image (717,844 33x21), image: ImagePool.Arrow black left
    Image (768,566 7x50), image: ImagePool.PipeBlack_1_Vertical
    Image (765,556 10x10), image: ImagePool.PipeBlack_1_LD
    Image (714,556 51x7), image: ImagePool.PipeBlack_1_Horizontal
    Image (704,581 10x11), image: ImagePool.PipeBlack_1_RU
    Image (704,499 7x84), image: ImagePool.PipeBlack_1_Vertical
    Image (704,489 10x10), image: ImagePool.PipeBlack_1_RD
    Image (711,489 19x7), image: ImagePool.PipeBlack_1_Horizontal
    Image (697,506 21x33), image: ImagePool.Arrow black down
    Image (714,585 28x7), image: ImagePool.PipeBlack_1_Horizontal
    Image (739,585 10x10), image: ImagePool.PipeBlack_1_LD
    Image (742,595 7x21), image: ImagePool.PipeBlack_1_Vertical
    Image (592,595 243x137), image: ImagePool.OilReceiver
    Image (400,135 314x7), image: ImagePool.PipeBlack_1_Horizontal
    Label (630,604 80x22), "Oil recevier"
    Image (522,553 7x296), image: ImagePool.PipeBlack_1_Vertical
    Image (519,544 10x10), image: ImagePool.PipeBlack_1_LD
    Image (400,544 120x7), image: ImagePool.PipeBlack_1_Horizontal
    Image (391,540 10x11), image: ImagePool.PipeBlack_1_RU
    Image (391,142 7x400), image: ImagePool.PipeBlack_1_Vertical
    Image (663,552 10x11), image: ImagePool.PipeBlack_1_RU
    Image (663,301 7x253), image: ImagePool.PipeBlack_1_Vertical
    Image (663,294 10x10), image: ImagePool.PipeBlack_1_RD
    Image (670,294 54x7), image: ImagePool.PipeBlack_1_Horizontal
    Image (656,383 21x33), image: ImagePool.Arrow black down
    Image (670,556 31x7), image: ImagePool.PipeBlack_1_Horizontal
    Image (727,241 7x53), image: ImagePool.PipeBlack_1_Vertical
    Image (724,290 10x11), image: ImagePool.PipeBlack_1_LU
    Image (757,380 10x10), image: ImagePool.PipeBlack_1_RD
    Image (764,380 22x7), image: ImagePool.PipeBlack_1_Horizontal
    Image (787,235 7x144), image: ImagePool.PipeBlack_1_Vertical
    Image (784,376 10x11), image: ImagePool.PipeBlack_1_LU
    Image (757,388 7x63), image: ImagePool.PipeBlack_1_Vertical
    Image (780,324 21x33), image: ImagePool.Arrow black down
    Label (750,471 80x22), "Ejector"
    Label (1223,551 80x22), "Evaporator"
    Image (384,339 21x33), image: ImagePool.Arrow black up
    Image (552,129 33x21), image: ImagePool.Arrow black right
    Image (360,529 232x131), image: ImagePool.OilFilter
    Label (379,561 59x22), "Oil filter"
    Line (987,843) (1025,821)
    Line (1100,816) (1116,807)
    Line (1004,817) (1102,761)
    Image (1097,823 38x38), image: ImagePool.RegValve
    Image (688,637 56x56), image: ImagePool.Pump_Large_3
    Polygon (710,660) (710,641) (734,663) (710,684) (710,676), colour toggle: Chiller_4.Comp_oil_pump
    Lamp1 (756,656 29x35), variable: Chiller_4.Oil_heater, style: Lamp-Lamp1-Green
    Label (744,683 55x22), "Heater"
    Image (1059,529 39x44), image: ImagePool.Valve_2
    Lamp1 (1066,529 24x25), variable: Chiller_4.Solenoid_oil_return, style: Lamp-Lamp1-Green
    Textfield (679,713 78x25), "%1.1f Hz", text variable: Chiller_4.Setpoint_conv_oil_pump
END_VISUALIZATION

(* text list Chiller_1_trendvalues (id | default)
  0 | Clear values
  1 | Chiller Capacity t1
  2 | dP CW
  3 | dP SW
  4 | Feedback Hot Gas Valve
  5 | Feedback Liquid Valve
  6 | Feedback PRV
  7 | Feedback Sea Water Valve
  8 | Feedback VGD
  9 | Hot Gas Valve Order
  10 | Liquid Level Condenser
  11 | Liquid Valve Order
  12 | Motor Current
  13 | Pressure CW Inlet
  14 | Pressure CW Outlet
  15 | Pressure Oil Compressor
  16 | Pressure Oil Diff
  17 | Pressure Oil Receiver
  18 | Pressure Suction Saturated
  19 | Pressure SW Inlet
  20 | Pressure SW Outlet
  21 | Sea Water Valve Order
  22 | Setpoint Liquid Level
  23 | Temp Chilled Medium Inlet
  24 | Temp Chilled Medium Outlet
  25 | Temp Discharge Gas
  26 | Temp Discharge Saturated
  27 | Temp Discharge Superheat
  28 | Temp Motor Air
  29 | Temp Motor Bearing DE
  30 | Temp Motor Bearing NDE
  31 | Temp Motor Winding R
  32 | Temp Motor Winding S
  33 | Temp Motor Winding T
  34 | Temp Oil Inlet Compressor
  35 | Temp Sea Water Inlet
  36 | Temp Suction Saturated
  37 | Temp Trafo Wind U
  38 | Temp Trafo Wind V
  39 | Temp Trafo Wind W
  40 | Theta Out
  41 | Thrust Bearing position
  42 | VFD Current Speed Hz
  43 | VFD Order Hz
   |  *)

(* text list Chiller_2_4_trendvalues (id | default)
  0 | Clear values
  1 | Chiller Capacity t1
  2 | dP CW
  3 | dP SW
  4 | Feedback Hot Gas Valve
  5 | Feedback Liquid Valve
  6 | Feedback PRV
  7 | Feedback Sea Water Valve
  8 | Hot Gas Valve Order
  9 | Liquid Level Condenser
  10 | Liquid Valve Order
  11 | Motor Current
  12 | Pressure CW Inlet
  13 | Pressure CW Outlet
  14 | Pressure Oil Compressor
  15 | Pressure Oil Diff
  16 | Pressure Oil Receiver
  17 | Pressure Suction Saturated
  18 | Pressure SW Inlet
  19 | Pressure SW Outlet
  20 | Sea Water Valve Order
  21 | Setpoint Liquid Level
  22 | Temp Chilled Medium Inlet
  23 | Temp Chilled Medium Outlet
  24 | Temp Discharge Gas
  25 | Temp Discharge Saturated
  26 | Temp Discharge Superheat
  27 | Temp Motor Air
  28 | Temp Motor Bearing DE
  29 | Temp Motor Bearing NDE
  30 | Temp Motor Winding R
  31 | Temp Motor Winding S
  32 | Temp Motor Winding T
  33 | Temp Oil Inlet Compressor
  34 | Temp Sea Water Inlet
  35 | Temp Suction Saturated
  36 | Theta Out
  37 | Thrust Bearing position
   |  *)

(* text list Chiller_3_trendvalues (id | default)
  0 | Clear values
  1 | Chiller Capacity t1
  2 | dP CW
  3 | dP SW
  4 | Feedback Hot Gas Valve
  5 | Feedback Liquid Valve
  6 | Feedback PRV
  7 | Feedback Sea Water Valve
  8 | Feedback VGD
  9 | Hot Gas Valve Order
  10 | Liquid Level Condenser
  11 | Liquid Valve Order
  12 | Motor Current
  13 | Pressure CW Inlet
  14 | Pressure CW Outlet
  15 | Pressure Oil Compressor
  16 | Pressure Oil Diff
  17 | Pressure Oil Receiver
  18 | Pressure Suction Saturated
  19 | Pressure SW Inlet
  20 | Pressure SW Outlet
  21 | Sea Water Valve Order
  22 | Setpoint Liquid Level
  23 | Temp Chilled Medium Inlet
  24 | Temp Chilled Medium Outlet
  25 | Temp Discharge Gas
  26 | Temp Discharge Saturated
  27 | Temp Discharge Superheat
  28 | Temp Motor Air
  29 | Temp Motor Bearing DE
  30 | Temp Motor Bearing NDE
  31 | Temp Motor Winding R
  32 | Temp Motor Winding S
  33 | Temp Motor Winding T
  34 | Temp Oil Inlet Compressor
  35 | Temp Sea Water Inlet
  36 | Temp Suction Saturated
  37 | Theta Out
  38 | Thrust Bearing position
   |  *)

(* text list Chiller_4_trendvalues (id | default)
  0 | Clear values
  1 | Chiller Capacity t1
  2 | dP CW
  3 | dP SW
  4 | Feedback Hot Gas Valve
  5 | Feedback Liquid Valve
  6 | Feedback PRV
  7 | Feedback Sea Water Valve
  8 | Hot Gas Valve Order
  9 | Liquid Level Condenser
  10 | Liquid Valve Order
  11 | Motor Current
  12 | Pressure CW Inlet
  13 | Pressure CW Outlet
  14 | Pressure Oil Compressor
  15 | Pressure Oil Diff
  16 | Pressure Oil Receiver
  17 | Pressure Suction Saturated
  18 | Pressure SW Inlet
  19 | Pressure SW Outlet
  20 | Sea Water Valve Order
  21 | Setpoint Liquid Level
  22 | Temp Chilled Medium Inlet
  23 | Temp Chilled Medium Outlet
  24 | Temp Discharge Gas
  25 | Temp Discharge Saturated
  26 | Temp Discharge Superheat
  27 | Temp Motor Air
  28 | Temp Motor Bearing DE
  29 | Temp Motor Bearing NDE
  30 | Temp Motor Winding R
  31 | Temp Motor Winding S
  32 | Temp Motor Winding T
  33 | Temp Oil Inlet Compressor
  34 | Temp Sea Water Inlet
  35 | Temp Suction Saturated
  36 | Theta Out
  37 | Thrust Bearing position
  38 | Feedback VGD
   |  *)

(* text list Sequence_trendvalues (id | default)
  0 | Clear values
  1 | Capacity Order AC1
  2 | Capacity Order AC2
  3 | Capacity Order AC3
  4 | Capacity Order AC4
  5 | COP ele AC1
  6 | COP ele AC2
  7 | COP ele AC3
  8 | COP ele AC4
  9 | P1 motor kW AC1
  10 | P1 motor kW AC2
  11 | P1 motor kW AC3
  12 | P1 motor kW AC4
  13 | Performance Index AC1
  14 | Performance Index AC2
  15 | Performance Index AC3
  16 | Performance Index AC4
  17 | Power Wasted AC1
  18 | Power Wasted AC2
  19 | Power Wasted AC3
  20 | Power Wasted AC4
  21 | Sequence Controller
  22 | Temp CW Delivery
  23 | Temp CW Return
  24 | Temp CW Setpoint
   |  *)

(* text PersistenceConfig
// Persistence configuration for application Device.Application
// Generated automatically by GenPersistence
SEC General
  Application := Device.Application ;
  ExcludedGroups := [  ] ;
  ToplevelInstanceNames := [ DataLogManager, PersistenceManager ] ;
  ToplevelFBPaths := [ GVL_DataLogManager.DataLogManager, GVL_PersistenceManager.PersistenceManager ] ;
END_SEC
SEC Channel : PersistenceChannel
  Groups := [ PersistenceChannel ] ;
  FBPath := PersistenceManager.INST_PersistenceChannel ;
  SeparateArchivePerToplevelInstance := False ;
  CompressTags := True ;
  MaximumFileSize := 0 ;
END_SEC
*)
